LIN {X 0,Y 523.924,Z 223.222,A -85,B 0,C 180,E1 -4895.227,E2 -4895.227} C_VEL
LIN {X 0,Y 523.919,Z 223.223,A -85,B 0,C 180,E1 -4898.102,E2 -4898.102} C_VEL
LIN {X 0,Y 523.938,Z 223.222,A -85,B 0,C 180,E1 -4901.093,E2 -4901.093} C_VEL
LIN {X 0,Y 523.927,Z 223.226,A -85,B 0,C 180,E1 -4904.23,E2 -4904.23} C_VEL
LIN {X 0,Y 523.894,Z 223.223,A -85,B 0,C 180,E1 -4906.898,E2 -4906.898} C_VEL
LIN {X 0,Y 523.235,Z 223.311,A -85,B 0,C 180,E1 -4907.54,E2 -4907.54} C_VEL
LIN {X 0,Y 520.406,Z 223.66,A -85,B 0,C 180,E1 -4908.581,E2 -4908.581} C_VEL
LIN {X 0,Y 518.008,Z 223.962,A -85,B 0,C 180,E1 -4909.421,E2 -4909.421} C_VEL
LIN {X 0,Y 516.973,Z 224.088,A -85,B 0,C 180,E1 -4910.068,E2 -4910.068} C_VEL
LIN {X 0,Y 516.886,Z 224.098,A -85,B 0,C 180,E1 -4910.288,E2 -4910.288} C_VEL
LIN {X 0,Y 516.849,Z 224.105,A -85,B 0,C 180,E1 -4913.348,E2 -4913.348} C_VEL
LIN {X 0,Y 516.656,Z 224.132,A -85,B 0,C 180,E1 -4916.102,E2 -4916.102} C_VEL
LIN {X 0,Y 516.569,Z 225.057,A -85,B 0,C 180,E1 -4917.514,E2 -4917.514} C_VEL
LIN {X 0,Y 516.551,Z 227.399,A -85,B 0,C 180,E1 -4919.774,E2 -4919.774} C_VEL
LIN {X 0,Y 516.547,Z 230.185,A -85,B 0,C 180,E1 -4922.445,E2 -4922.445} C_VEL
LIN {X 0,Y 516.449,Z 232.938,A -85,B 0,C 180,E1 -4925.048,E2 -4925.048} C_VEL
LIN {X 0,Y 516.412,Z 235.802,A -85,B 0,C 180,E1 -4927.734,E2 -4927.734} C_VEL
LIN {X 0,Y 516.339,Z 239.349,A -85,B 0,C 180,E1 -4930.933,E2 -4930.933} C_VEL
LIN {X 0,Y 516.316,Z 242.204,A -85,B 0,C 180,E1 -4933.39,E2 -4933.39} C_VEL
LIN {X 0,Y 516.364,Z 245.681,A -85,B 0,C 180,E1 -4936.195,E2 -4936.195} C_VEL
LIN {X 0,Y 518.536,Z 256.766,A -85,B 0,C 180,E1 -4936.554,E2 -4936.554} C_VEL
LIN {X 0,Y 518.351,Z 269.23,A -85,B 0,C 180,E1 -4937.023,E2 -4937.023} C_VEL
LIN {X 0,Y 518.082,Z 280.828,A -85,B 0,C 180,E1 -4937.612,E2 -4937.612} C_VEL
LIN {X 0,Y 517.755,Z 292.099,A -85,B 0,C 180,E1 -4938.351,E2 -4938.351} C_VEL
LIN {X 0,Y 517.448,Z 302.758,A -85,B 0,C 180,E1 -4939.236,E2 -4939.236} C_VEL
LIN {X 0,Y 517.179,Z 312.341,A -85,B 0,C 180,E1 -4940.22,E2 -4940.22} C_VEL
LIN {X 0,Y 516.938,Z 320.187,A -85,B 0,C 180,E1 -4941.202,E2 -4941.202} C_VEL
LIN {X 0,Y 516.709,Z 327.857,A -85,B 0,C 180,E1 -4942.379,E2 -4942.379} C_VEL
LIN {X 0,Y 516.547,Z 334.883,A -85,B 0,C 180,E1 -4943.751,E2 -4943.751} C_VEL
LIN {X 0,Y 516.38,Z 339.568,A -85,B 0,C 180,E1 -4944.925,E2 -4944.925} C_VEL
LIN {X 0,Y 516.374,Z 343.149,A -85,B 0,C 180,E1 -4946.098,E2 -4946.098} C_VEL
LIN {X 0,Y 516.363,Z 345.001,A -85,B 0,C 180,E1 -4946.879,E2 -4946.879} C_VEL
LIN {X 0,Y 516.264,Z 346.404,A -85,B 0,C 180,E1 -4947.659,E2 -4947.659} C_VEL
LIN {X 0,Y 516.182,Z 348.013,A -85,B 0,C 180,E1 -4949.22,E2 -4949.22} C_VEL
LIN {X 0,Y 516.181,Z 348.249,A -85,B 0,C 180,E1 -4950,E2 -4950} C_VEL
LIN {X 0,Y 516.181,Z 348.067,A -85,B 0,C 180,E1 -4950.78,E2 -4950.78} C_VEL
LIN {X 0,Y 516.264,Z 346.529,A -85,B 0,C 180,E1 -4952.34,E2 -4952.34} C_VEL
LIN {X 0,Y 516.363,Z 345.18,A -85,B 0,C 180,E1 -4953.121,E2 -4953.121} C_VEL
LIN {X 0,Y 516.384,Z 342.34,A -85,B 0,C 180,E1 -4954.293,E2 -4954.293} C_VEL
LIN {X 0,Y 516.405,Z 338.488,A -85,B 0,C 180,E1 -4955.467,E2 -4955.467} C_VEL
LIN {X 0,Y 516.543,Z 333.377,A -85,B 0,C 180,E1 -4956.67,E2 -4956.67} C_VEL
LIN {X 0,Y 516.729,Z 327.242,A -85,B 0,C 180,E1 -4957.817,E2 -4957.817} C_VEL
LIN {X 0,Y 516.934,Z 319.392,A -85,B 0,C 180,E1 -4958.995,E2 -4958.995} C_VEL
LIN {X 0,Y 517.189,Z 311.383,A -85,B 0,C 180,E1 -4959.977,E2 -4959.977} C_VEL
LIN {X 0,Y 517.467,Z 301.605,A -85,B 0,C 180,E1 -4960.961,E2 -4960.961} C_VEL
LIN {X 0,Y 517.781,Z 291.979,A -85,B 0,C 180,E1 -4961.747,E2 -4961.747} C_VEL
LIN {X 0,Y 518.035,Z 281.52,A -85,B 0,C 180,E1 -4962.44,E2 -4962.44} C_VEL
LIN {X 0,Y 518.341,Z 269.027,A -85,B 0,C 180,E1 -4963.077,E2 -4963.077} C_VEL
LIN {X 0,Y 518.392,Z 255.726,A -85,B 0,C 180,E1 -4963.575,E2 -4963.575} C_VEL
LIN {X 0,Y 516.333,Z 245.547,A -85,B 0,C 180,E1 -4963.906,E2 -4963.906} C_VEL
LIN {X 0,Y 516.348,Z 242.346,A -85,B 0,C 180,E1 -4966.608,E2 -4966.608} C_VEL
LIN {X 0,Y 516.34,Z 239.456,A -85,B 0,C 180,E1 -4969.067,E2 -4969.067} C_VEL
LIN {X 0,Y 516.411,Z 235.882,A -85,B 0,C 180,E1 -4972.265,E2 -4972.265} C_VEL
LIN {X 0,Y 516.448,Z 232.99,A -85,B 0,C 180,E1 -4974.952,E2 -4974.952} C_VEL
LIN {X 0,Y 516.522,Z 229.994,A -85,B 0,C 180,E1 -4977.82,E2 -4977.82} C_VEL
LIN {X 0,Y 516.574,Z 226.678,A -85,B 0,C 180,E1 -4981.005,E2 -4981.005} C_VEL
LIN {X 0,Y 516.584,Z 224.643,A -85,B 0,C 180,E1 -4982.969,E2 -4982.969} C_VEL
LIN {X 0,Y 516.647,Z 224.133,A -85,B 0,C 180,E1 -4983.923,E2 -4983.923} C_VEL
LIN {X 0,Y 516.85,Z 224.105,A -85,B 0,C 180,E1 -4986.749,E2 -4986.749} C_VEL
LIN {X 0,Y 516.885,Z 224.098,A -85,B 0,C 180,E1 -4989.721,E2 -4989.721} C_VEL
LIN {X 0,Y 516.909,Z 224.096,A -85,B 0,C 180,E1 -4991.776,E2 -4991.776} C_VEL
LIN {X 0,Y 516.898,Z 224.095,A -85,B 0,C 180,E1 -4995.007,E2 -4995.007} C_VEL
LIN {X 0,Y 516.905,Z 224.096,A -85,B 0,C 180,E1 -4998.4,E2 -4998.4} C_VEL
LIN {X 0,Y 516.883,Z 224.101,A -85,B 0,C 180,E1 -5001.284,E2 -5001.284} C_VEL
LIN {X 0,Y 516.874,Z 224.104,A -85,B 0,C 180,E1 -5004.22,E2 -5004.22} C_VEL
LIN {X 0,Y 516.884,Z 224.098,A -85,B 0,C 180,E1 -5007.052,E2 -5007.052} C_VEL
LIN {X 0,Y 516.867,Z 224.102,A -85,B 0,C 180,E1 -5009.794,E2 -5009.794} C_VEL
LIN {X 0,Y 516.886,Z 224.1,A -85,B 0,C 180,E1 -5012.465,E2 -5012.465} C_VEL
LIN {X 0,Y 516.871,Z 224.101,A -85,B 0,C 180,E1 -5015.07,E2 -5015.07} C_VEL
LIN {X 0,Y 516.872,Z 224.103,A -85,B 0,C 180,E1 -5017.622,E2 -5017.622} C_VEL
LIN {X 0,Y 516.932,Z 224.093,A -85,B 0,C 180,E1 -5020.13,E2 -5020.13} C_VEL
LIN {X 0,Y 516.876,Z 224.101,A -85,B 0,C 180,E1 -5023.409,E2 -5023.409} C_VEL
LIN {X 0,Y 516.875,Z 224.099,A -85,B 0,C 180,E1 -5025.833,E2 -5025.833} C_VEL
LIN {X 0,Y 516.97,Z 224.091,A -85,B 0,C 180,E1 -5028.234,E2 -5028.234} C_VEL
LIN {X 0,Y 516.969,Z 224.092,A -85,B 0,C 180,E1 -5031.4,E2 -5031.4} C_VEL
LIN {X 0,Y 517.003,Z 224.085,A -85,B 0,C 180,E1 -5033.757,E2 -5033.757} C_VEL
LIN {X 0,Y 516.98,Z 224.09,A -85,B 0,C 180,E1 -5036.883,E2 -5036.883} C_VEL
LIN {X 0,Y 516.962,Z 224.093,A -85,B 0,C 180,E1 -5038.442,E2 -5038.442} C_VEL
LIN {X 0,Y 517.093,Z 224.073,A -85,B 0,C 180,E1 -5040.779,E2 -5040.779} C_VEL
LIN {X 0,Y 517.014,Z 224.084,A -85,B 0,C 180,E1 -5043.117,E2 -5043.117} C_VEL
LIN {X 0,Y 517.006,Z 224.084,A -85,B 0,C 180,E1 -5046.243,E2 -5046.243} C_VEL
LIN {X 0,Y 516.935,Z 224.091,A -85,B 0,C 180,E1 -5049.39,E2 -5049.39} C_VEL
LIN {X 0,Y 516.902,Z 224.097,A -85,B 0,C 180,E1 -5052.565,E2 -5052.565} C_VEL
LIN {X 0,Y 516.903,Z 224.1,A -85,B 0,C 180,E1 -5055.779,E2 -5055.779} C_VEL
LIN {X 0,Y 516.928,Z 224.093,A -85,B 0,C 180,E1 -5058.222,E2 -5058.222} C_VEL
LIN {X 0,Y 516.916,Z 224.097,A -85,B 0,C 180,E1 -5060.701,E2 -5060.701} C_VEL
LIN {X 0,Y 516.886,Z 224.103,A -85,B 0,C 180,E1 -5064.073,E2 -5064.073} C_VEL
LIN {X 0,Y 516.841,Z 224.102,A -85,B 0,C 180,E1 -5066.663,E2 -5066.663} C_VEL
LIN {X 0,Y 516.889,Z 224.101,A -85,B 0,C 180,E1 -5069.519,E2 -5069.519} C_VEL
LIN {X 0,Y 516.899,Z 224.099,A -85,B 0,C 180,E1 -5072.543,E2 -5072.543} C_VEL
LIN {X 0,Y 516.867,Z 224.101,A -85,B 0,C 180,E1 -5075.329,E2 -5075.329} C_VEL
LIN {X 0,Y 516.879,Z 224.101,A -85,B 0,C 180,E1 -5077.942,E2 -5077.942} C_VEL
LIN {X 0,Y 516.852,Z 224.102,A -85,B 0,C 180,E1 -5080.745,E2 -5080.745} C_VEL
LIN {X 0,Y 516.883,Z 224.098,A -85,B 0,C 180,E1 -5083.903,E2 -5083.903} C_VEL
LIN {X 0,Y 516.884,Z 224.103,A -85,B 0,C 180,E1 -5086.107,E2 -5086.107} C_VEL
LIN {X 0,Y 516.916,Z 224.098,A -85,B 0,C 180,E1 -5088.399,E2 -5088.399} C_VEL
LIN {X 0,Y 516.895,Z 224.105,A -85,B 0,C 180,E1 -5091.385,E2 -5091.385} C_VEL
LIN {X 0,Y 518.007,Z 230.529,A -85,B 0,C 180,E1 -5093.83,E2 -5093.83} C_VEL
LIN {X 0,Y 518.034,Z 237.244,A -85,B 0,C 180,E1 -5096.204,E2 -5096.204} C_VEL
LIN {X 0,Y 517.77,Z 245.421,A -85,B 0,C 180,E1 -5098.949,E2 -5098.949} C_VEL
LIN {X 0,Y 517.573,Z 254.625,A -85,B 0,C 180,E1 -5101.96,E2 -5101.96} C_VEL
LIN {X 0,Y 517.321,Z 262.957,A -85,B 0,C 180,E1 -5104.663,E2 -5104.663} C_VEL
LIN {X 0,Y 517.117,Z 272.225,A -85,B 0,C 180,E1 -5107.633,E2 -5107.633} C_VEL
LIN {X 0,Y 516.906,Z 281.492,A -85,B 0,C 180,E1 -5110.542,E2 -5110.542} C_VEL
LIN {X 0,Y 516.71,Z 290.759,A -85,B 0,C 180,E1 -5113.403,E2 -5113.403} C_VEL
LIN {X 0,Y 516.582,Z 299.732,A -85,B 0,C 180,E1 -5116.095,E2 -5116.095} C_VEL
LIN {X 0,Y 518.513,Z 312.183,A -85,B 0,C 180,E1 -5116.429,E2 -5116.429} C_VEL
LIN {X 0,Y 518.281,Z 324.984,A -85,B 0,C 180,E1 -5116.872,E2 -5116.872} C_VEL
LIN {X 0,Y 517.947,Z 337.175,A -85,B 0,C 180,E1 -5117.461,E2 -5117.461} C_VEL
LIN {X 0,Y 517.652,Z 347.772,A -85,B 0,C 180,E1 -5118.122,E2 -5118.122} C_VEL
LIN {X 0,Y 517.411,Z 358.262,A -85,B 0,C 180,E1 -5118.939,E2 -5118.939} C_VEL
LIN {X 0,Y 517.093,Z 367.539,A -85,B 0,C 180,E1 -5119.823,E2 -5119.823} C_VEL
LIN {X 0,Y 516.867,Z 375.991,A -85,B 0,C 180,E1 -5120.807,E2 -5120.807} C_VEL
LIN {X 0,Y 516.641,Z 384.237,A -85,B 0,C 180,E1 -5121.985,E2 -5121.985} C_VEL
LIN {X 0,Y 516.479,Z 391.077,A -85,B 0,C 180,E1 -5123.201,E2 -5123.201} C_VEL
LIN {X 0,Y 516.405,Z 396.95,A -85,B 0,C 180,E1 -5124.533,E2 -5124.533} C_VEL
LIN {X 0,Y 516.344,Z 400.895,A -85,B 0,C 180,E1 -5125.707,E2 -5125.707} C_VEL
LIN {X 0,Y 516.282,Z 403.808,A -85,B 0,C 180,E1 -5126.879,E2 -5126.879} C_VEL
LIN {X 0,Y 516.261,Z 405.197,A -85,B 0,C 180,E1 -5127.659,E2 -5127.659} C_VEL
LIN {X 0,Y 516.16,Z 406.786,A -85,B 0,C 180,E1 -5129.22,E2 -5129.22} C_VEL
LIN {X 0,Y 516.154,Z 407,A -85,B 0,C 180,E1 -5130,E2 -5130} C_VEL
LIN {X 0,Y 516.192,Z 406.185,A -85,B 0,C 180,E1 -5131.56,E2 -5131.56} C_VEL
LIN {X 0,Y 516.261,Z 405.198,A -85,B 0,C 180,E1 -5132.341,E2 -5132.341} C_VEL
LIN {X 0,Y 516.282,Z 403.81,A -85,B 0,C 180,E1 -5133.121,E2 -5133.121} C_VEL
LIN {X 0,Y 516.344,Z 400.895,A -85,B 0,C 180,E1 -5134.293,E2 -5134.293} C_VEL
LIN {X 0,Y 516.405,Z 396.948,A -85,B 0,C 180,E1 -5135.467,E2 -5135.467} C_VEL
LIN {X 0,Y 516.487,Z 391.03,A -85,B 0,C 180,E1 -5136.808,E2 -5136.808} C_VEL
LIN {X 0,Y 516.641,Z 384.236,A -85,B 0,C 180,E1 -5138.015,E2 -5138.015} C_VEL
LIN {X 0,Y 516.868,Z 375.99,A -85,B 0,C 180,E1 -5139.194,E2 -5139.194} C_VEL
LIN {X 0,Y 517.093,Z 367.537,A -85,B 0,C 180,E1 -5140.177,E2 -5140.177} C_VEL
LIN {X 0,Y 517.453,Z 357.094,A -85,B 0,C 180,E1 -5141.16,E2 -5141.16} C_VEL
LIN {X 0,Y 517.706,Z 345.73,A -85,B 0,C 180,E1 -5142.019,E2 -5142.019} C_VEL
LIN {X 0,Y 517.987,Z 335.404,A -85,B 0,C 180,E1 -5142.638,E2 -5142.638} C_VEL
LIN {X 0,Y 518.294,Z 323.758,A -85,B 0,C 180,E1 -5143.178,E2 -5143.178} C_VEL
LIN {X 0,Y 518.436,Z 310.796,A -85,B 0,C 180,E1 -5143.611,E2 -5143.611} C_VEL
LIN {X 0,Y 516.566,Z 299.529,A -85,B 0,C 180,E1 -5143.925,E2 -5143.925} C_VEL
LIN {X 0,Y 516.71,Z 290.759,A -85,B 0,C 180,E1 -5146.597,E2 -5146.597} C_VEL
LIN {X 0,Y 516.906,Z 281.491,A -85,B 0,C 180,E1 -5149.458,E2 -5149.458} C_VEL
LIN {X 0,Y 517.1,Z 271.962,A -85,B 0,C 180,E1 -5152.452,E2 -5152.452} C_VEL
LIN {X 0,Y 517.322,Z 262.957,A -85,B 0,C 180,E1 -5155.337,E2 -5155.337} C_VEL
LIN {X 0,Y 517.574,Z 254.625,A -85,B 0,C 180,E1 -5158.04,E2 -5158.04} C_VEL
LIN {X 0,Y 517.805,Z 244.879,A -85,B 0,C 180,E1 -5161.231,E2 -5161.231} C_VEL
LIN {X 0,Y 518.051,Z 236.209,A -85,B 0,C 180,E1 -5164.153,E2 -5164.153} C_VEL
LIN {X 0,Y 518.005,Z 230.494,A -85,B 0,C 180,E1 -5166.17,E2 -5166.17} C_VEL
LIN {X 0,Y 516.889,Z 224.104,A -85,B 0,C 180,E1 -5168.616,E2 -5168.616} C_VEL
LIN {X 0,Y 516.915,Z 224.101,A -85,B 0,C 180,E1 -5171.775,E2 -5171.775} C_VEL
LIN {X 0,Y 516.899,Z 224.101,A -85,B 0,C 180,E1 -5175.007,E2 -5175.007} C_VEL
LIN {X 0,Y 516.889,Z 224.098,A -85,B 0,C 180,E1 -5178.402,E2 -5178.402} C_VEL
LIN {X 0,Y 516.877,Z 224.098,A -85,B 0,C 180,E1 -5181.284,E2 -5181.284} C_VEL
LIN {X 0,Y 516.872,Z 224.104,A -85,B 0,C 180,E1 -5184.22,E2 -5184.22} C_VEL
LIN {X 0,Y 516.899,Z 224.1,A -85,B 0,C 180,E1 -5187.053,E2 -5187.053} C_VEL
LIN {X 0,Y 516.871,Z 224.1,A -85,B 0,C 180,E1 -5189.795,E2 -5189.795} C_VEL
LIN {X 0,Y 516.876,Z 224.105,A -85,B 0,C 180,E1 -5192.464,E2 -5192.464} C_VEL
LIN {X 0,Y 516.847,Z 224.102,A -85,B 0,C 180,E1 -5195.069,E2 -5195.069} C_VEL
LIN {X 0,Y 516.874,Z 224.103,A -85,B 0,C 180,E1 -5197.622,E2 -5197.622} C_VEL
LIN {X 0,Y 516.937,Z 224.092,A -85,B 0,C 180,E1 -5200.13,E2 -5200.13} C_VEL
LIN {X 0,Y 516.912,Z 224.099,A -85,B 0,C 180,E1 -5202.596,E2 -5202.596} C_VEL
LIN {X 0,Y 516.94,Z 224.092,A -85,B 0,C 180,E1 -5205.03,E2 -5205.03} C_VEL
LIN {X 0,Y 516.93,Z 224.093,A -85,B 0,C 180,E1 -5208.233,E2 -5208.233} C_VEL
LIN {X 0,Y 516.951,Z 224.095,A -85,B 0,C 180,E1 -5211.399,E2 -5211.399} C_VEL
LIN {X 0,Y 517.007,Z 224.083,A -85,B 0,C 180,E1 -5213.757,E2 -5213.757} C_VEL
LIN {X 0,Y 517.015,Z 224.084,A -85,B 0,C 180,E1 -5216.883,E2 -5216.883} C_VEL
LIN {X 0,Y 517.095,Z 224.072,A -85,B 0,C 180,E1 -5219.221,E2 -5219.221} C_VEL
LIN {X 0,Y 517.075,Z 224.073,A -85,B 0,C 180,E1 -5222.337,E2 -5222.337} C_VEL
LIN {X 0,Y 517.026,Z 224.082,A -85,B 0,C 180,E1 -5225.46,E2 -5225.46} C_VEL
LIN {X 0,Y 516.968,Z 224.089,A -85,B 0,C 180,E1 -5227.813,E2 -5227.813} C_VEL
LIN {X 0,Y 516.956,Z 224.09,A -85,B 0,C 180,E1 -5230.972,E2 -5230.972} C_VEL
LIN {X 0,Y 516.906,Z 224.1,A -85,B 0,C 180,E1 -5233.364,E2 -5233.364} C_VEL
LIN {X 0,Y 516.858,Z 224.101,A -85,B 0,C 180,E1 -5235.781,E2 -5235.781} C_VEL
LIN {X 0,Y 516.883,Z 224.098,A -85,B 0,C 180,E1 -5238.224,E2 -5238.224} C_VEL
LIN {X 0,Y 516.918,Z 224.097,A -85,B 0,C 180,E1 -5240.701,E2 -5240.701} C_VEL
LIN {X 0,Y 516.896,Z 224.101,A -85,B 0,C 180,E1 -5244.073,E2 -5244.073} C_VEL
LIN {X 0,Y 516.915,Z 224.095,A -85,B 0,C 180,E1 -5246.659,E2 -5246.659} C_VEL
LIN {X 0,Y 516.884,Z 224.098,A -85,B 0,C 180,E1 -5249.517,E2 -5249.517} C_VEL
LIN {X 0,Y 516.899,Z 224.1,A -85,B 0,C 180,E1 -5252.543,E2 -5252.543} C_VEL
LIN {X 0,Y 516.87,Z 224.101,A -85,B 0,C 180,E1 -5255.329,E2 -5255.329} C_VEL
LIN {X 0,Y 516.884,Z 224.1,A -85,B 0,C 180,E1 -5257.943,E2 -5257.943} C_VEL
LIN {X 0,Y 516.885,Z 224.103,A -85,B 0,C 180,E1 -5260.742,E2 -5260.742} C_VEL
LIN {X 0,Y 516.884,Z 224.099,A -85,B 0,C 180,E1 -5263.903,E2 -5263.903} C_VEL
LIN {X 0,Y 516.848,Z 224.101,A -85,B 0,C 180,E1 -5266.899,E2 -5266.899} C_VEL
LIN {X 0,Y 516.884,Z 224.103,A -85,B 0,C 180,E1 -5269.59,E2 -5269.59} C_VEL
LIN {X 0,Y 516.886,Z 224.098,A -85,B 0,C 180,E1 -5270.288,E2 -5270.288} C_VEL
LIN {X 0,Y 516.213,Z 224.184,A -85,B 0,C 180,E1 -5270.938,E2 -5270.938} C_VEL
LIN {X 0,Y 513.361,Z 224.539,A -85,B 0,C 180,E1 -5271.993,E2 -5271.993} C_VEL
LIN {X 0,Y 510.939,Z 224.842,A -85,B 0,C 180,E1 -5272.843,E2 -5272.843} C_VEL
LIN {X 0,Y 509.878,Z 224.972,A -85,B 0,C 180,E1 -5273.5,E2 -5273.5} C_VEL
LIN {X 0,Y 509.781,Z 224.984,A -85,B 0,C 180,E1 -5273.722,E2 -5273.722} C_VEL
LIN {X 0,Y 509.56,Z 225.014,A -85,B 0,C 180,E1 -5276.516,E2 -5276.516} C_VEL
LIN {X 0,Y 509.513,Z 227.071,A -85,B 0,C 180,E1 -5278.782,E2 -5278.782} C_VEL
LIN {X 0,Y 509.466,Z 230.42,A -85,B 0,C 180,E1 -5282.029,E2 -5282.029} C_VEL
LIN {X 0,Y 509.405,Z 233.186,A -85,B 0,C 180,E1 -5284.679,E2 -5284.679} C_VEL
LIN {X 0,Y 509.326,Z 236.28,A -85,B 0,C 180,E1 -5287.595,E2 -5287.595} C_VEL
LIN {X 0,Y 509.265,Z 239.624,A -85,B 0,C 180,E1 -5290.658,E2 -5290.658} C_VEL
LIN {X 0,Y 509.254,Z 242.514,A -85,B 0,C 180,E1 -5293.153,E2 -5293.153} C_VEL
LIN {X 0,Y 509.325,Z 246.006,A -85,B 0,C 180,E1 -5296.001,E2 -5296.001} C_VEL
LIN {X 0,Y 511.642,Z 257.212,A -85,B 0,C 180,E1 -5296.369,E2 -5296.369} C_VEL
LIN {X 0,Y 511.447,Z 269.671,A -85,B 0,C 180,E1 -5296.844,E2 -5296.844} C_VEL
LIN {X 0,Y 511.16,Z 281.811,A -85,B 0,C 180,E1 -5297.472,E2 -5297.472} C_VEL
LIN {X 0,Y 510.832,Z 292.533,A -85,B 0,C 180,E1 -5298.191,E2 -5298.191} C_VEL
LIN {X 0,Y 510.493,Z 303.191,A -85,B 0,C 180,E1 -5299.088,E2 -5299.088} C_VEL
LIN {X 0,Y 510.193,Z 312.774,A -85,B 0,C 180,E1 -5300.085,E2 -5300.085} C_VEL
LIN {X 0,Y 509.95,Z 320.618,A -85,B 0,C 180,E1 -5301.08,E2 -5301.08} C_VEL
LIN {X 0,Y 509.67,Z 328.288,A -85,B 0,C 180,E1 -5302.273,E2 -5302.273} C_VEL
LIN {X 0,Y 509.501,Z 335.312,A -85,B 0,C 180,E1 -5303.664,E2 -5303.664} C_VEL
LIN {X 0,Y 509.311,Z 339.998,A -85,B 0,C 180,E1 -5304.854,E2 -5304.854} C_VEL
LIN {X 0,Y 509.308,Z 343.578,A -85,B 0,C 180,E1 -5306.044,E2 -5306.044} C_VEL
LIN {X 0,Y 509.304,Z 345.428,A -85,B 0,C 180,E1 -5306.836,E2 -5306.836} C_VEL
LIN {X 0,Y 509.195,Z 346.831,A -85,B 0,C 180,E1 -5307.627,E2 -5307.627} C_VEL
LIN {X 0,Y 509.096,Z 348.44,A -85,B 0,C 180,E1 -5309.209,E2 -5309.209} C_VEL
LIN {X 0,Y 509.095,Z 348.676,A -85,B 0,C 180,E1 -5310,E2 -5310} C_VEL
LIN {X 0,Y 509.095,Z 348.494,A -85,B 0,C 180,E1 -5310.791,E2 -5310.791} C_VEL
LIN {X 0,Y 509.195,Z 346.954,A -85,B 0,C 180,E1 -5312.373,E2 -5312.373} C_VEL
LIN {X 0,Y 509.304,Z 345.605,A -85,B 0,C 180,E1 -5313.164,E2 -5313.164} C_VEL
LIN {X 0,Y 509.32,Z 342.765,A -85,B 0,C 180,E1 -5314.352,E2 -5314.352} C_VEL
LIN {X 0,Y 509.35,Z 338.913,A -85,B 0,C 180,E1 -5315.543,E2 -5315.543} C_VEL
LIN {X 0,Y 509.509,Z 333.083,A -85,B 0,C 180,E1 -5316.91,E2 -5316.91} C_VEL
LIN {X 0,Y 509.738,Z 326.449,A -85,B 0,C 180,E1 -5318.124,E2 -5318.124} C_VEL
LIN {X 0,Y 509.969,Z 318.344,A -85,B 0,C 180,E1 -5319.319,E2 -5319.319} C_VEL
LIN {X 0,Y 510.305,Z 310.036,A -85,B 0,C 180,E1 -5320.314,E2 -5320.314} C_VEL
LIN {X 0,Y 510.602,Z 299.779,A -85,B 0,C 180,E1 -5321.311,E2 -5321.311} C_VEL
LIN {X 0,Y 510.956,Z 288.483,A -85,B 0,C 180,E1 -5322.188,E2 -5322.188} C_VEL
LIN {X 0,Y 511.283,Z 276.667,A -85,B 0,C 180,E1 -5322.907,E2 -5322.907} C_VEL
LIN {X 0,Y 511.529,Z 264.673,A -85,B 0,C 180,E1 -5323.457,E2 -5323.457} C_VEL
LIN {X 0,Y 511.478,Z 256.521,A -85,B 0,C 180,E1 -5323.749,E2 -5323.749} C_VEL
LIN {X 0,Y 509.289,Z 245.909,A -85,B 0,C 180,E1 -5324.102,E2 -5324.102} C_VEL
LIN {X 0,Y 509.278,Z 242.62,A -85,B 0,C 180,E1 -5326.846,E2 -5326.846} C_VEL
LIN {X 0,Y 509.265,Z 239.73,A -85,B 0,C 180,E1 -5329.342,E2 -5329.342} C_VEL
LIN {X 0,Y 509.324,Z 236.364,A -85,B 0,C 180,E1 -5332.404,E2 -5332.404} C_VEL
LIN {X 0,Y 509.404,Z 233.253,A -85,B 0,C 180,E1 -5335.321,E2 -5335.321} C_VEL
LIN {X 0,Y 509.453,Z 230.472,A -85,B 0,C 180,E1 -5338.006,E2 -5338.006} C_VEL
LIN {X 0,Y 509.512,Z 227.14,A -85,B 0,C 180,E1 -5341.217,E2 -5341.217} C_VEL
LIN {X 0,Y 509.557,Z 225.015,A -85,B 0,C 180,E1 -5343.484,E2 -5343.484} C_VEL
LIN {X 0,Y 509.785,Z 224.983,A -85,B 0,C 180,E1 -5346.357,E2 -5346.357} C_VEL
LIN {X 0,Y 509.849,Z 224.977,A -85,B 0,C 180,E1 -5349.352,E2 -5349.352} C_VEL
LIN {X 0,Y 509.816,Z 224.981,A -85,B 0,C 180,E1 -5352.492,E2 -5352.492} C_VEL
LIN {X 0,Y 509.841,Z 224.976,A -85,B 0,C 180,E1 -5355.33,E2 -5355.33} C_VEL
LIN {X 0,Y 509.848,Z 224.976,A -85,B 0,C 180,E1 -5358.573,E2 -5358.573} C_VEL
LIN {X 0,Y 509.853,Z 224.975,A -85,B 0,C 180,E1 -5361.787,E2 -5361.787} C_VEL
LIN {X 0,Y 509.833,Z 224.978,A -85,B 0,C 180,E1 -5364.622,E2 -5364.622} C_VEL
LIN {X 0,Y 509.863,Z 224.976,A -85,B 0,C 180,E1 -5367.481,E2 -5367.481} C_VEL
LIN {X 0,Y 509.855,Z 224.973,A -85,B 0,C 180,E1 -5370.275,E2 -5370.275} C_VEL
LIN {X 0,Y 509.882,Z 224.971,A -85,B 0,C 180,E1 -5373.629,E2 -5373.629} C_VEL
LIN {X 0,Y 509.826,Z 224.98,A -85,B 0,C 180,E1 -5376.436,E2 -5376.436} C_VEL
LIN {X 0,Y 509.92,Z 224.968,A -85,B 0,C 180,E1 -5379.845,E2 -5379.845} C_VEL
LIN {X 0,Y 509.849,Z 224.979,A -85,B 0,C 180,E1 -5383.173,E2 -5383.173} C_VEL
LIN {X 0,Y 509.848,Z 224.974,A -85,B 0,C 180,E1 -5385.634,E2 -5385.634} C_VEL
LIN {X 0,Y 509.917,Z 224.967,A -85,B 0,C 180,E1 -5388.875,E2 -5388.875} C_VEL
LIN {X 0,Y 509.954,Z 224.963,A -85,B 0,C 180,E1 -5392.078,E2 -5392.078} C_VEL
LIN {X 0,Y 509.977,Z 224.959,A -85,B 0,C 180,E1 -5394.464,E2 -5394.464} C_VEL
LIN {X 0,Y 510.044,Z 224.948,A -85,B 0,C 180,E1 -5397.631,E2 -5397.631} C_VEL
LIN {X 0,Y 510.064,Z 224.948,A -85,B 0,C 180,E1 -5400.789,E2 -5400.789} C_VEL
LIN {X 0,Y 509.956,Z 224.964,A -85,B 0,C 180,E1 -5403.16,E2 -5403.16} C_VEL
LIN {X 0,Y 509.957,Z 224.962,A -85,B 0,C 180,E1 -5406.33,E2 -5406.33} C_VEL
LIN {X 0,Y 509.902,Z 224.972,A -85,B 0,C 180,E1 -5408.72,E2 -5408.72} C_VEL
LIN {X 0,Y 509.903,Z 224.97,A -85,B 0,C 180,E1 -5411.932,E2 -5411.932} C_VEL
LIN {X 0,Y 509.898,Z 224.97,A -85,B 0,C 180,E1 -5415.242,E2 -5415.242} C_VEL
LIN {X 0,Y 509.886,Z 224.971,A -85,B 0,C 180,E1 -5417.998,E2 -5417.998} C_VEL
LIN {X 0,Y 509.854,Z 224.977,A -85,B 0,C 180,E1 -5421.002,E2 -5421.002} C_VEL
LIN {X 0,Y 509.821,Z 224.979,A -85,B 0,C 180,E1 -5423.564,E2 -5423.564} C_VEL
LIN {X 0,Y 509.817,Z 224.978,A -85,B 0,C 180,E1 -5426.356,E2 -5426.356} C_VEL
LIN {X 0,Y 509.839,Z 224.977,A -85,B 0,C 180,E1 -5428.847,E2 -5428.847} C_VEL
LIN {X 0,Y 509.821,Z 224.979,A -85,B 0,C 180,E1 -5431.59,E2 -5431.59} C_VEL
LIN {X 0,Y 509.849,Z 224.977,A -85,B 0,C 180,E1 -5434.414,E2 -5434.414} C_VEL
LIN {X 0,Y 509.809,Z 224.981,A -85,B 0,C 180,E1 -5437.342,E2 -5437.342} C_VEL
LIN {X 0,Y 509.815,Z 224.977,A -85,B 0,C 180,E1 -5440.385,E2 -5440.385} C_VEL
LIN {X 0,Y 509.801,Z 224.985,A -85,B 0,C 180,E1 -5443.059,E2 -5443.059} C_VEL
LIN {X 0,Y 509.824,Z 224.979,A -85,B 0,C 180,E1 -5445.793,E2 -5445.793} C_VEL
LIN {X 0,Y 509.858,Z 224.977,A -85,B 0,C 180,E1 -5448.574,E2 -5448.574} C_VEL
LIN {X 0,Y 509.853,Z 225.045,A -85,B 0,C 180,E1 -5451.157,E2 -5451.157} C_VEL
LIN {X 0,Y 511.032,Z 231.69,A -85,B 0,C 180,E1 -5453.746,E2 -5453.746} C_VEL
LIN {X 0,Y 511.089,Z 237.083,A -85,B 0,C 180,E1 -5455.681,E2 -5455.681} C_VEL
LIN {X 0,Y 510.847,Z 245.392,A -85,B 0,C 180,E1 -5458.536,E2 -5458.536} C_VEL
LIN {X 0,Y 510.561,Z 255.093,A -85,B 0,C 180,E1 -5461.761,E2 -5461.761} C_VEL
LIN {X 0,Y 510.3,Z 264.281,A -85,B 0,C 180,E1 -5464.726,E2 -5464.726} C_VEL
LIN {X 0,Y 510.081,Z 273.672,A -85,B 0,C 180,E1 -5467.774,E2 -5467.774} C_VEL
LIN {X 0,Y 509.856,Z 282.816,A -85,B 0,C 180,E1 -5470.681,E2 -5470.681} C_VEL
LIN {X 0,Y 509.645,Z 293.407,A -85,B 0,C 180,E1 -5473.99,E2 -5473.99} C_VEL
LIN {X 0,Y 509.536,Z 299.731,A -85,B 0,C 180,E1 -5475.899,E2 -5475.899} C_VEL
LIN {X 0,Y 511.588,Z 312.183,A -85,B 0,C 180,E1 -5476.241,E2 -5476.241} C_VEL
LIN {X 0,Y 511.361,Z 324.984,A -85,B 0,C 180,E1 -5476.691,E2 -5476.691} C_VEL
LIN {X 0,Y 511.024,Z 337.174,A -85,B 0,C 180,E1 -5477.288,E2 -5477.288} C_VEL
LIN {X 0,Y 510.674,Z 348.197,A -85,B 0,C 180,E1 -5477.987,E2 -5477.987} C_VEL
LIN {X 0,Y 510.371,Z 359.4,A -85,B 0,C 180,E1 -5478.885,E2 -5478.885} C_VEL
LIN {X 0,Y 510.035,Z 369.335,A -85,B 0,C 180,E1 -5479.881,E2 -5479.881} C_VEL
LIN {X 0,Y 509.76,Z 378.961,A -85,B 0,C 180,E1 -5481.077,E2 -5481.077} C_VEL
LIN {X 0,Y 509.522,Z 386.622,A -85,B 0,C 180,E1 -5482.271,E2 -5482.271} C_VEL
LIN {X 0,Y 509.336,Z 393.68,A -85,B 0,C 180,E1 -5483.662,E2 -5483.662} C_VEL
LIN {X 0,Y 509.248,Z 398.373,A -85,B 0,C 180,E1 -5484.853,E2 -5484.853} C_VEL
LIN {X 0,Y 509.253,Z 401.958,A -85,B 0,C 180,E1 -5486.043,E2 -5486.043} C_VEL
LIN {X 0,Y 509.2,Z 403.808,A -85,B 0,C 180,E1 -5486.835,E2 -5486.835} C_VEL
LIN {X 0,Y 509.161,Z 405.196,A -85,B 0,C 180,E1 -5487.627,E2 -5487.627} C_VEL
LIN {X 0,Y 509.073,Z 406.786,A -85,B 0,C 180,E1 -5489.209,E2 -5489.209} C_VEL
LIN {X 0,Y 509.065,Z 407,A -85,B 0,C 180,E1 -5490,E2 -5490} C_VEL
LIN {X 0,Y 509.112,Z 406.185,A -85,B 0,C 180,E1 -5491.582,E2 -5491.582} C_VEL
LIN {X 0,Y 509.161,Z 405.198,A -85,B 0,C 180,E1 -5492.373,E2 -5492.373} C_VEL
LIN {X 0,Y 509.2,Z 403.81,A -85,B 0,C 180,E1 -5493.165,E2 -5493.165} C_VEL
LIN {X 0,Y 509.234,Z 400.895,A -85,B 0,C 180,E1 -5494.353,E2 -5494.353} C_VEL
LIN {X 0,Y 509.345,Z 396.948,A -85,B 0,C 180,E1 -5495.543,E2 -5495.543} C_VEL
LIN {X 0,Y 509.41,Z 391.281,A -85,B 0,C 180,E1 -5496.854,E2 -5496.854} C_VEL
LIN {X 0,Y 509.585,Z 384.235,A -85,B 0,C 180,E1 -5498.127,E2 -5498.127} C_VEL
LIN {X 0,Y 509.846,Z 375.99,A -85,B 0,C 180,E1 -5499.321,E2 -5499.321} C_VEL
LIN {X 0,Y 510.083,Z 367.537,A -85,B 0,C 180,E1 -5500.318,E2 -5500.318} C_VEL
LIN {X 0,Y 510.479,Z 357.093,A -85,B 0,C 180,E1 -5501.314,E2 -5501.314} C_VEL
LIN {X 0,Y 510.738,Z 346.472,A -85,B 0,C 180,E1 -5502.133,E2 -5502.133} C_VEL
LIN {X 0,Y 511.054,Z 335.404,A -85,B 0,C 180,E1 -5502.812,E2 -5502.812} C_VEL
LIN {X 0,Y 511.396,Z 323.758,A -85,B 0,C 180,E1 -5503.359,E2 -5503.359} C_VEL
LIN {X 0,Y 511.527,Z 311.71,A -85,B 0,C 180,E1 -5503.773,E2 -5503.773} C_VEL
LIN {X 0,Y 509.526,Z 299.529,A -85,B 0,C 180,E1 -5504.121,E2 -5504.121} C_VEL
LIN {X 0,Y 509.718,Z 289.435,A -85,B 0,C 180,E1 -5507.244,E2 -5507.244} C_VEL
LIN {X 0,Y 509.948,Z 279.334,A -85,B 0,C 180,E1 -5510.419,E2 -5510.419} C_VEL
LIN {X 0,Y 510.178,Z 269.576,A -85,B 0,C 180,E1 -5513.547,E2 -5513.547} C_VEL
LIN {X 0,Y 510.429,Z 260.488,A -85,B 0,C 180,E1 -5516.495,E2 -5516.495} C_VEL
LIN {X 0,Y 510.585,Z 252.003,A -85,B 0,C 180,E1 -5519.252,E2 -5519.252} C_VEL
LIN {X 0,Y 510.878,Z 243.878,A -85,B 0,C 180,E1 -5521.981,E2 -5521.981} C_VEL
LIN {X 0,Y 511.114,Z 235.729,A -85,B 0,C 180,E1 -5524.795,E2 -5524.795} C_VEL
LIN {X 0,Y 511.029,Z 231.678,A -85,B 0,C 180,E1 -5526.254,E2 -5526.254} C_VEL
LIN {X 0,Y 509.856,Z 224.979,A -85,B 0,C 180,E1 -5528.907,E2 -5528.907} C_VEL
LIN {X 0,Y 509.859,Z 224.98,A -85,B 0,C 180,E1 -5531.897,E2 -5531.897} C_VEL
LIN {X 0,Y 509.843,Z 224.978,A -85,B 0,C 180,E1 -5534.67,E2 -5534.67} C_VEL
LIN {X 0,Y 509.808,Z 224.981,A -85,B 0,C 180,E1 -5537.507,E2 -5537.507} C_VEL
LIN {X 0,Y 509.834,Z 224.981,A -85,B 0,C 180,E1 -5540.646,E2 -5540.646} C_VEL
LIN {X 0,Y 509.813,Z 224.981,A -85,B 0,C 180,E1 -5543.646,E2 -5543.646} C_VEL
LIN {X 0,Y 509.863,Z 224.973,A -85,B 0,C 180,E1 -5546.539,E2 -5546.539} C_VEL
LIN {X 0,Y 509.838,Z 224.978,A -85,B 0,C 180,E1 -5549.334,E2 -5549.334} C_VEL
LIN {X 0,Y 509.835,Z 224.977,A -85,B 0,C 180,E1 -5552.051,E2 -5552.051} C_VEL
LIN {X 0,Y 509.803,Z 224.98,A -85,B 0,C 180,E1 -5554.7,E2 -5554.7} C_VEL
LIN {X 0,Y 509.83,Z 224.979,A -85,B 0,C 180,E1 -5557.458,E2 -5557.458} C_VEL
LIN {X 0,Y 509.922,Z 224.967,A -85,B 0,C 180,E1 -5559.845,E2 -5559.845} C_VEL
LIN {X 0,Y 509.878,Z 224.973,A -85,B 0,C 180,E1 -5563.174,E2 -5563.174} C_VEL
LIN {X 0,Y 509.855,Z 224.974,A -85,B 0,C 180,E1 -5565.634,E2 -5565.634} C_VEL
LIN {X 0,Y 509.894,Z 224.971,A -85,B 0,C 180,E1 -5568.131,E2 -5568.131} C_VEL
LIN {X 0,Y 509.897,Z 224.972,A -85,B 0,C 180,E1 -5571.279,E2 -5571.279} C_VEL
LIN {X 0,Y 509.959,Z 224.962,A -85,B 0,C 180,E1 -5573.67,E2 -5573.67} C_VEL
LIN {X 0,Y 510.06,Z 224.95,A -85,B 0,C 180,E1 -5577.631,E2 -5577.631} C_VEL
LIN {X 0,Y 510.038,Z 224.954,A -85,B 0,C 180,E1 -5580,E2 -5580} C_VEL
LIN {X 0,Y 510.046,Z 224.948,A -85,B 0,C 180,E1 -5582.369,E2 -5582.369} C_VEL
LIN {X 0,Y 509.956,Z 224.963,A -85,B 0,C 180,E1 -5586.33,E2 -5586.33} C_VEL
LIN {X 0,Y 509.909,Z 224.971,A -85,B 0,C 180,E1 -5588.72,E2 -5588.72} C_VEL
LIN {X 0,Y 509.91,Z 224.97,A -85,B 0,C 180,E1 -5591.932,E2 -5591.932} C_VEL
LIN {X 0,Y 509.9,Z 224.973,A -85,B 0,C 180,E1 -5595.242,E2 -5595.242} C_VEL
LIN {X 0,Y 509.843,Z 224.977,A -85,B 0,C 180,E1 -5598.485,E2 -5598.485} C_VEL
LIN {X 0,Y 509.856,Z 224.975,A -85,B 0,C 180,E1 -5601.002,E2 -5601.002} C_VEL
LIN {X 0,Y 509.828,Z 224.98,A -85,B 0,C 180,E1 -5603.564,E2 -5603.564} C_VEL
LIN {X 0,Y 509.911,Z 224.967,A -85,B 0,C 180,E1 -5606.377,E2 -5606.377} C_VEL
LIN {X 0,Y 509.83,Z 224.976,A -85,B 0,C 180,E1 -5609.753,E2 -5609.753} C_VEL
LIN {X 0,Y 509.871,Z 224.973,A -85,B 0,C 180,E1 -5612.773,E2 -5612.773} C_VEL
LIN {X 0,Y 509.83,Z 224.979,A -85,B 0,C 180,E1 -5615.578,E2 -5615.578} C_VEL
LIN {X 0,Y 509.854,Z 224.975,A -85,B 0,C 180,E1 -5618.338,E2 -5618.338} C_VEL
LIN {X 0,Y 509.855,Z 224.975,A -85,B 0,C 180,E1 -5621.426,E2 -5621.426} C_VEL
LIN {X 0,Y 509.843,Z 224.976,A -85,B 0,C 180,E1 -5624.67,E2 -5624.67} C_VEL
LIN {X 0,Y 509.848,Z 224.977,A -85,B 0,C 180,E1 -5628.105,E2 -5628.105} C_VEL
LIN {X 0,Y 509.85,Z 224.976,A -85,B 0,C 180,E1 -5630.647,E2 -5630.647} C_VEL
LIN {X 0,Y 509.788,Z 224.983,A -85,B 0,C 180,E1 -5633.643,E2 -5633.643} C_VEL
LIN {X 0,Y 509.781,Z 224.984,A -85,B 0,C 180,E1 -5633.722,E2 -5633.722} C_VEL
LIN {X 0,Y 509.064,Z 225.096,A -85,B 0,C 180,E1 -5634.382,E2 -5634.382} C_VEL
LIN {X 0,Y 506.114,Z 225.445,A -85,B 0,C 180,E1 -5635.452,E2 -5635.452} C_VEL
LIN {X 0,Y 503.631,Z 225.753,A -85,B 0,C 180,E1 -5636.313,E2 -5636.313} C_VEL
LIN {X 0,Y 502.551,Z 225.984,A -85,B 0,C 180,E1 -5636.977,E2 -5636.977} C_VEL
LIN {X 0,Y 502.455,Z 226.166,A -85,B 0,C 180,E1 -5637.201,E2 -5637.201} C_VEL
LIN {X 0,Y 502.428,Z 229.16,A -85,B 0,C 180,E1 -5640.142,E2 -5640.142} C_VEL
LIN {X 0,Y 502.363,Z 231.604,A -85,B 0,C 180,E1 -5642.505,E2 -5642.505} C_VEL
LIN {X 0,Y 502.292,Z 234.649,A -85,B 0,C 180,E1 -5645.433,E2 -5645.433} C_VEL
LIN {X 0,Y 502.253,Z 237.144,A -85,B 0,C 180,E1 -5647.802,E2 -5647.802} C_VEL
LIN {X 0,Y 502.212,Z 239.931,A -85,B 0,C 180,E1 -5650.375,E2 -5650.375} C_VEL
LIN {X 0,Y 502.214,Z 242.826,A -85,B 0,C 180,E1 -5652.91,E2 -5652.91} C_VEL
LIN {X 0,Y 502.227,Z 246.326,A -85,B 0,C 180,E1 -5655.799,E2 -5655.799} C_VEL
LIN {X 0,Y 504.767,Z 258.416,A -85,B 0,C 180,E1 -5656.206,E2 -5656.206} C_VEL
LIN {X 0,Y 504.558,Z 271.235,A -85,B 0,C 180,E1 -5656.713,E2 -5656.713} C_VEL
LIN {X 0,Y 504.254,Z 282.668,A -85,B 0,C 180,E1 -5657.323,E2 -5657.323} C_VEL
LIN {X 0,Y 503.86,Z 294.25,A -85,B 0,C 180,E1 -5658.127,E2 -5658.127} C_VEL
LIN {X 0,Y 503.519,Z 304.685,A -85,B 0,C 180,E1 -5659.037,E2 -5659.037} C_VEL
LIN {X 0,Y 503.222,Z 313.206,A -85,B 0,C 180,E1 -5659.946,E2 -5659.946} C_VEL
LIN {X 0,Y 502.949,Z 321.049,A -85,B 0,C 180,E1 -5660.955,E2 -5660.955} C_VEL
LIN {X 0,Y 502.642,Z 328.719,A -85,B 0,C 180,E1 -5662.165,E2 -5662.165} C_VEL
LIN {X 0,Y 502.455,Z 335.742,A -85,B 0,C 180,E1 -5663.575,E2 -5663.575} C_VEL
LIN {X 0,Y 502.244,Z 340.428,A -85,B 0,C 180,E1 -5664.781,E2 -5664.781} C_VEL
LIN {X 0,Y 502.245,Z 344.006,A -85,B 0,C 180,E1 -5665.988,E2 -5665.988} C_VEL
LIN {X 0,Y 502.246,Z 345.855,A -85,B 0,C 180,E1 -5666.791,E2 -5666.791} C_VEL
LIN {X 0,Y 502.13,Z 347.258,A -85,B 0,C 180,E1 -5667.593,E2 -5667.593} C_VEL
LIN {X 0,Y 502.011,Z 348.867,A -85,B 0,C 180,E1 -5669.198,E2 -5669.198} C_VEL
LIN {X 0,Y 502.008,Z 349.103,A -85,B 0,C 180,E1 -5670,E2 -5670} C_VEL
LIN {X 0,Y 502.011,Z 348.92,A -85,B 0,C 180,E1 -5670.802,E2 -5670.802} C_VEL
LIN {X 0,Y 502.13,Z 347.379,A -85,B 0,C 180,E1 -5672.406,E2 -5672.406} C_VEL
LIN {X 0,Y 502.247,Z 346.03,A -85,B 0,C 180,E1 -5673.209,E2 -5673.209} C_VEL
LIN {X 0,Y 502.259,Z 343.19,A -85,B 0,C 180,E1 -5674.414,E2 -5674.414} C_VEL
LIN {X 0,Y 502.297,Z 339.337,A -85,B 0,C 180,E1 -5675.621,E2 -5675.621} C_VEL
LIN {X 0,Y 502.478,Z 333.7,A -85,B 0,C 180,E1 -5676.968,E2 -5676.968} C_VEL
LIN {X 0,Y 502.707,Z 326.873,A -85,B 0,C 180,E1 -5678.239,E2 -5678.239} C_VEL
LIN {X 0,Y 502.968,Z 318.766,A -85,B 0,C 180,E1 -5679.45,E2 -5679.45} C_VEL
LIN {X 0,Y 503.347,Z 310.457,A -85,B 0,C 180,E1 -5680.458,E2 -5680.458} C_VEL
LIN {X 0,Y 503.668,Z 300.198,A -85,B 0,C 180,E1 -5681.469,E2 -5681.469} C_VEL
LIN {X 0,Y 504.02,Z 289.386,A -85,B 0,C 180,E1 -5682.324,E2 -5682.324} C_VEL
LIN {X 0,Y 504.36,Z 278.892,A -85,B 0,C 180,E1 -5682.985,E2 -5682.985} C_VEL
LIN {X 0,Y 504.638,Z 266.377,A -85,B 0,C 180,E1 -5683.592,E2 -5683.592} C_VEL
LIN {X 0,Y 504.558,Z 257.311,A -85,B 0,C 180,E1 -5683.928,E2 -5683.928} C_VEL
LIN {X 0,Y 502.223,Z 246.264,A -85,B 0,C 180,E1 -5684.305,E2 -5684.305} C_VEL
LIN {X 0,Y 502.231,Z 242.933,A -85,B 0,C 180,E1 -5687.089,E2 -5687.089} C_VEL
LIN {X 0,Y 502.243,Z 239.212,A -85,B 0,C 180,E1 -5690.356,E2 -5690.356} C_VEL
LIN {X 0,Y 502.25,Z 236.302,A -85,B 0,C 180,E1 -5693.067,E2 -5693.067} C_VEL
LIN {X 0,Y 502.325,Z 233.517,A -85,B 0,C 180,E1 -5695.704,E2 -5695.704} C_VEL
LIN {X 0,Y 502.401,Z 230.746,A -85,B 0,C 180,E1 -5698.4,E2 -5698.4} C_VEL
LIN {X 0,Y 502.466,Z 227.641,A -85,B 0,C 180,E1 -5701.437,E2 -5701.437} C_VEL
LIN {X 0,Y 502.464,Z 225.998,A -85,B 0,C 180,E1 -5703.059,E2 -5703.059} C_VEL
LIN {X 0,Y 502.739,Z 225.863,A -85,B 0,C 180,E1 -5705.954,E2 -5705.954} C_VEL
LIN {X 0,Y 502.804,Z 225.855,A -85,B 0,C 180,E1 -5708.976,E2 -5708.976} C_VEL
LIN {X 0,Y 502.806,Z 225.857,A -85,B 0,C 180,E1 -5712.199,E2 -5712.199} C_VEL
LIN {X 0,Y 502.788,Z 225.855,A -85,B 0,C 180,E1 -5715.47,E2 -5715.47} C_VEL
LIN {X 0,Y 502.797,Z 225.855,A -85,B 0,C 180,E1 -5717.861,E2 -5717.861} C_VEL
LIN {X 0,Y 502.802,Z 225.855,A -85,B 0,C 180,E1 -5721.024,E2 -5721.024} C_VEL
LIN {X 0,Y 502.778,Z 225.86,A -85,B 0,C 180,E1 -5724.169,E2 -5724.169} C_VEL
LIN {X 0,Y 502.833,Z 225.848,A -85,B 0,C 180,E1 -5726.994,E2 -5726.994} C_VEL
LIN {X 0,Y 502.812,Z 225.851,A -85,B 0,C 180,E1 -5730.066,E2 -5730.066} C_VEL
LIN {X 0,Y 502.847,Z 225.848,A -85,B 0,C 180,E1 -5733.444,E2 -5733.444} C_VEL
LIN {X 0,Y 502.779,Z 225.858,A -85,B 0,C 180,E1 -5736.085,E2 -5736.085} C_VEL
LIN {X 0,Y 502.787,Z 225.855,A -85,B 0,C 180,E1 -5738.689,E2 -5738.689} C_VEL
LIN {X 0,Y 502.815,Z 225.855,A -85,B 0,C 180,E1 -5741.248,E2 -5741.248} C_VEL
LIN {X 0,Y 502.838,Z 225.851,A -85,B 0,C 180,E1 -5744.665,E2 -5744.665} C_VEL
LIN {X 0,Y 502.88,Z 225.845,A -85,B 0,C 180,E1 -5748.039,E2 -5748.039} C_VEL
LIN {X 0,Y 502.875,Z 225.846,A -85,B 0,C 180,E1 -5751.157,E2 -5751.157} C_VEL
LIN {X 0,Y 502.908,Z 225.841,A -85,B 0,C 180,E1 -5753.581,E2 -5753.581} C_VEL
LIN {X 0,Y 502.868,Z 225.849,A -85,B 0,C 180,E1 -5756.795,E2 -5756.795} C_VEL
LIN {X 0,Y 502.9,Z 225.844,A -85,B 0,C 180,E1 -5758.398,E2 -5758.398} C_VEL
LIN {X 0,Y 503.014,Z 225.827,A -85,B 0,C 180,E1 -5760.801,E2 -5760.801} C_VEL
LIN {X 0,Y 502.899,Z 225.843,A -85,B 0,C 180,E1 -5763.204,E2 -5763.204} C_VEL
LIN {X 0,Y 502.91,Z 225.84,A -85,B 0,C 180,E1 -5766.419,E2 -5766.419} C_VEL
LIN {X 0,Y 502.861,Z 225.847,A -85,B 0,C 180,E1 -5768.844,E2 -5768.844} C_VEL
LIN {X 0,Y 502.845,Z 225.852,A -85,B 0,C 180,E1 -5772.102,E2 -5772.102} C_VEL
LIN {X 0,Y 502.852,Z 225.848,A -85,B 0,C 180,E1 -5775.4,E2 -5775.4} C_VEL
LIN {X 0,Y 502.844,Z 225.848,A -85,B 0,C 180,E1 -5778.12,E2 -5778.12} C_VEL
LIN {X 0,Y 502.832,Z 225.852,A -85,B 0,C 180,E1 -5780.536,E2 -5780.536} C_VEL
LIN {X 0,Y 502.789,Z 225.854,A -85,B 0,C 180,E1 -5783.041,E2 -5783.041} C_VEL
LIN {X 0,Y 502.778,Z 225.859,A -85,B 0,C 180,E1 -5785.679,E2 -5785.679} C_VEL
LIN {X 0,Y 502.775,Z 225.855,A -85,B 0,C 180,E1 -5788.377,E2 -5788.377} C_VEL
LIN {X 0,Y 502.795,Z 225.858,A -85,B 0,C 180,E1 -5791.143,E2 -5791.143} C_VEL
LIN {X 0,Y 502.806,Z 225.855,A -85,B 0,C 180,E1 -5793.994,E2 -5793.994} C_VEL
LIN {X 0,Y 502.766,Z 225.858,A -85,B 0,C 180,E1 -5797.176,E2 -5797.176} C_VEL
LIN {X 0,Y 502.772,Z 225.855,A -85,B 0,C 180,E1 -5800.017,E2 -5800.017} C_VEL
LIN {X 0,Y 502.773,Z 225.855,A -85,B 0,C 180,E1 -5802.195,E2 -5802.195} C_VEL
LIN {X 0,Y 502.788,Z 225.855,A -85,B 0,C 180,E1 -5805.47,E2 -5805.47} C_VEL
LIN {X 0,Y 502.822,Z 225.852,A -85,B 0,C 180,E1 -5808.934,E2 -5808.934} C_VEL
LIN {X 0,Y 502.818,Z 225.93,A -85,B 0,C 180,E1 -5810.896,E2 -5810.896} C_VEL
LIN {X 0,Y 504.008,Z 232.701,A -85,B 0,C 180,E1 -5813.601,E2 -5813.601} C_VEL
LIN {X 0,Y 504.111,Z 238.544,A -85,B 0,C 180,E1 -5815.724,E2 -5815.724} C_VEL
LIN {X 0,Y 503.774,Z 247.738,A -85,B 0,C 180,E1 -5818.924,E2 -5818.924} C_VEL
LIN {X 0,Y 503.508,Z 257.283,A -85,B 0,C 180,E1 -5822.122,E2 -5822.122} C_VEL
LIN {X 0,Y 503.276,Z 265.479,A -85,B 0,C 180,E1 -5824.792,E2 -5824.792} C_VEL
LIN {X 0,Y 503.026,Z 274.872,A -85,B 0,C 180,E1 -5827.838,E2 -5827.838} C_VEL
LIN {X 0,Y 502.8,Z 284.14,A -85,B 0,C 180,E1 -5830.824,E2 -5830.824} C_VEL
LIN {X 0,Y 502.561,Z 294.731,A -85,B 0,C 180,E1 -5834.175,E2 -5834.175} C_VEL
LIN {X 0,Y 502.482,Z 299.582,A -85,B 0,C 180,E1 -5835.693,E2 -5835.693} C_VEL
LIN {X 0,Y 504.688,Z 313.096,A -85,B 0,C 180,E1 -5836.075,E2 -5836.075} C_VEL
LIN {X 0,Y 504.424,Z 326.112,A -85,B 0,C 180,E1 -5836.556,E2 -5836.556} C_VEL
LIN {X 0,Y 504.036,Z 338.643,A -85,B 0,C 180,E1 -5837.194,E2 -5837.194} C_VEL
LIN {X 0,Y 503.694,Z 349.589,A -85,B 0,C 180,E1 -5837.919,E2 -5837.919} C_VEL
LIN {X 0,Y 503.359,Z 360.47,A -85,B 0,C 180,E1 -5838.83,E2 -5838.83} C_VEL
LIN {X 0,Y 503.032,Z 369.334,A -85,B 0,C 180,E1 -5839.739,E2 -5839.739} C_VEL
LIN {X 0,Y 502.704,Z 378.961,A -85,B 0,C 180,E1 -5840.951,E2 -5840.951} C_VEL
LIN {X 0,Y 502.47,Z 386.622,A -85,B 0,C 180,E1 -5842.162,E2 -5842.162} C_VEL
LIN {X 0,Y 502.275,Z 393.68,A -85,B 0,C 180,E1 -5843.573,E2 -5843.573} C_VEL
LIN {X 0,Y 502.185,Z 398.373,A -85,B 0,C 180,E1 -5844.781,E2 -5844.781} C_VEL
LIN {X 0,Y 502.151,Z 401.958,A -85,B 0,C 180,E1 -5845.987,E2 -5845.987} C_VEL
LIN {X 0,Y 502.121,Z 403.808,A -85,B 0,C 180,E1 -5846.791,E2 -5846.791} C_VEL
LIN {X 0,Y 502.066,Z 405.195,A -85,B 0,C 180,E1 -5847.593,E2 -5847.593} C_VEL
LIN {X 0,Y 501.99,Z 406.786,A -85,B 0,C 180,E1 -5849.198,E2 -5849.198} C_VEL
LIN {X 0,Y 501.98,Z 407,A -85,B 0,C 180,E1 -5850,E2 -5850} C_VEL
LIN {X 0,Y 502.036,Z 406.185,A -85,B 0,C 180,E1 -5851.605,E2 -5851.605} C_VEL
LIN {X 0,Y 502.066,Z 405.197,A -85,B 0,C 180,E1 -5852.407,E2 -5852.407} C_VEL
LIN {X 0,Y 502.121,Z 403.81,A -85,B 0,C 180,E1 -5853.21,E2 -5853.21} C_VEL
LIN {X 0,Y 502.128,Z 400.895,A -85,B 0,C 180,E1 -5854.415,E2 -5854.415} C_VEL
LIN {X 0,Y 502.26,Z 396.948,A -85,B 0,C 180,E1 -5855.621,E2 -5855.621} C_VEL
LIN {X 0,Y 502.336,Z 390.976,A -85,B 0,C 180,E1 -5857.012,E2 -5857.012} C_VEL
LIN {X 0,Y 502.542,Z 384.235,A -85,B 0,C 180,E1 -5858.242,E2 -5858.242} C_VEL
LIN {X 0,Y 502.811,Z 375.99,A -85,B 0,C 180,E1 -5859.453,E2 -5859.453} C_VEL
LIN {X 0,Y 503.077,Z 367.537,A -85,B 0,C 180,E1 -5860.464,E2 -5860.464} C_VEL
LIN {X 0,Y 503.505,Z 357.092,A -85,B 0,C 180,E1 -5861.473,E2 -5861.473} C_VEL
LIN {X 0,Y 503.799,Z 345.382,A -85,B 0,C 180,E1 -5862.381,E2 -5862.381} C_VEL
LIN {X 0,Y 504.172,Z 333.485,A -85,B 0,C 180,E1 -5863.092,E2 -5863.092} C_VEL
LIN {X 0,Y 504.541,Z 321.161,A -85,B 0,C 180,E1 -5863.647,E2 -5863.647} C_VEL
LIN {X 0,Y 504.546,Z 312.167,A -85,B 0,C 180,E1 -5863.955,E2 -5863.955} C_VEL
LIN {X 0,Y 502.465,Z 299.529,A -85,B 0,C 180,E1 -5864.324,E2 -5864.324} C_VEL
LIN {X 0,Y 502.663,Z 289.435,A -85,B 0,C 180,E1 -5867.494,E2 -5867.494} C_VEL
LIN {X 0,Y 502.905,Z 279.828,A -85,B 0,C 180,E1 -5870.558,E2 -5870.558} C_VEL
LIN {X 0,Y 503.188,Z 269.576,A -85,B 0,C 180,E1 -5873.894,E2 -5873.894} C_VEL
LIN {X 0,Y 503.454,Z 259.907,A -85,B 0,C 180,E1 -5877.012,E2 -5877.012} C_VEL
LIN {X 0,Y 503.724,Z 250.436,A -85,B 0,C 180,E1 -5880.151,E2 -5880.151} C_VEL
LIN {X 0,Y 504.012,Z 241.57,A -85,B 0,C 180,E1 -5883.212,E2 -5883.212} C_VEL
LIN {X 0,Y 504.168,Z 234.188,A -85,B 0,C 180,E1 -5885.837,E2 -5885.837} C_VEL
LIN {X 0,Y 503.335,Z 228.864,A -85,B 0,C 180,E1 -5887.906,E2 -5887.906} C_VEL
LIN {X 0,Y 502.802,Z 225.857,A -85,B 0,C 180,E1 -5889.17,E2 -5889.17} C_VEL
LIN {X 0,Y 502.807,Z 225.858,A -85,B 0,C 180,E1 -5892.199,E2 -5892.199} C_VEL
LIN {X 0,Y 502.789,Z 225.859,A -85,B 0,C 180,E1 -5895.47,E2 -5895.47} C_VEL
LIN {X 0,Y 502.798,Z 225.852,A -85,B 0,C 180,E1 -5897.861,E2 -5897.861} C_VEL
LIN {X 0,Y 502.795,Z 225.854,A -85,B 0,C 180,E1 -5901.023,E2 -5901.023} C_VEL
LIN {X 0,Y 502.775,Z 225.86,A -85,B 0,C 180,E1 -5904.17,E2 -5904.17} C_VEL
LIN {X 0,Y 502.837,Z 225.851,A -85,B 0,C 180,E1 -5906.994,E2 -5906.994} C_VEL
LIN {X 0,Y 502.814,Z 225.851,A -85,B 0,C 180,E1 -5910.066,E2 -5910.066} C_VEL
LIN {X 0,Y 502.777,Z 225.854,A -85,B 0,C 180,E1 -5913.46,E2 -5913.46} C_VEL
LIN {X 0,Y 502.771,Z 225.861,A -85,B 0,C 180,E1 -5916.085,E2 -5916.085} C_VEL
LIN {X 0,Y 502.788,Z 225.855,A -85,B 0,C 180,E1 -5918.689,E2 -5918.689} C_VEL
LIN {X 0,Y 502.832,Z 225.852,A -85,B 0,C 180,E1 -5921.248,E2 -5921.248} C_VEL
LIN {X 0,Y 502.854,Z 225.848,A -85,B 0,C 180,E1 -5924.6,E2 -5924.6} C_VEL
LIN {X 0,Y 502.874,Z 225.847,A -85,B 0,C 180,E1 -5928.043,E2 -5928.043} C_VEL
LIN {X 0,Y 502.856,Z 225.848,A -85,B 0,C 180,E1 -5931.156,E2 -5931.156} C_VEL
LIN {X 0,Y 502.911,Z 225.84,A -85,B 0,C 180,E1 -5933.581,E2 -5933.581} C_VEL
LIN {X 0,Y 502.9,Z 225.843,A -85,B 0,C 180,E1 -5936.796,E2 -5936.796} C_VEL
LIN {X 0,Y 503.015,Z 225.826,A -85,B 0,C 180,E1 -5939.199,E2 -5939.199} C_VEL
LIN {X 0,Y 503.015,Z 225.824,A -85,B 0,C 180,E1 -5942.402,E2 -5942.402} C_VEL
LIN {X 0,Y 502.933,Z 225.837,A -85,B 0,C 180,E1 -5945.614,E2 -5945.614} C_VEL
LIN {X 0,Y 502.886,Z 225.845,A -85,B 0,C 180,E1 -5948.034,E2 -5948.034} C_VEL
LIN {X 0,Y 502.882,Z 225.844,A -85,B 0,C 180,E1 -5951.283,E2 -5951.283} C_VEL
LIN {X 0,Y 502.83,Z 225.849,A -85,B 0,C 180,E1 -5954.571,E2 -5954.571} C_VEL
LIN {X 0,Y 502.806,Z 225.85,A -85,B 0,C 180,E1 -5957.909,E2 -5957.909} C_VEL
LIN {X 0,Y 502.834,Z 225.853,A -85,B 0,C 180,E1 -5960.536,E2 -5960.536} C_VEL
LIN {X 0,Y 502.793,Z 225.854,A -85,B 0,C 180,E1 -5963.041,E2 -5963.041} C_VEL
LIN {X 0,Y 502.824,Z 225.852,A -85,B 0,C 180,E1 -5965.677,E2 -5965.677} C_VEL
LIN {X 0,Y 502.777,Z 225.856,A -85,B 0,C 180,E1 -5968.377,E2 -5968.377} C_VEL
LIN {X 0,Y 502.795,Z 225.851,A -85,B 0,C 180,E1 -5971.498,E2 -5971.498} C_VEL
LIN {X 0,Y 502.794,Z 225.856,A -85,B 0,C 180,E1 -5973.995,E2 -5973.995} C_VEL
LIN {X 0,Y 502.782,Z 225.857,A -85,B 0,C 180,E1 -5977.178,E2 -5977.178} C_VEL
LIN {X 0,Y 502.791,Z 225.854,A -85,B 0,C 180,E1 -5980.015,E2 -5980.015} C_VEL
LIN {X 0,Y 502.807,Z 225.854,A -85,B 0,C 180,E1 -5982.199,E2 -5982.199} C_VEL
LIN {X 0,Y 502.789,Z 225.853,A -85,B 0,C 180,E1 -5985.47,E2 -5985.47} C_VEL
LIN {X 0,Y 502.798,Z 225.858,A -85,B 0,C 180,E1 -5987.86,E2 -5987.86} C_VEL
LIN {X 0,Y 502.805,Z 225.854,A -85,B 0,C 180,E1 -5991.024,E2 -5991.024} C_VEL
LIN {X 0,Y 502.74,Z 225.863,A -85,B 0,C 180,E1 -5994.175,E2 -5994.175} C_VEL
LIN {X 0,Y 502.465,Z 226.02,A -85,B 0,C 180,E1 -5997.059,E2 -5997.059} C_VEL
LIN {X 0,Y 502.455,Z 226.166,A -85,B 0,C 180,E1 -5997.201,E2 -5997.201} C_VEL
LIN {X 0,Y 501.764,Z 226.917,A -85,B 0,C 180,E1 -5997.865,E2 -5997.865} C_VEL
LIN {X 0,Y 498.887,Z 228.292,A -85,B 0,C 180,E1 -5998.939,E2 -5998.939} C_VEL
LIN {X 0,Y 496.461,Z 229.412,A -85,B 0,C 180,E1 -5999.805,E2 -5999.805} C_VEL
LIN {X 0,Y 495.414,Z 230.199,A -85,B 0,C 180,E1 -6000.475,E2 -6000.475} C_VEL
LIN {X 0,Y 495.324,Z 230.441,A -85,B 0,C 180,E1 -6000.702,E2 -6000.702} C_VEL
LIN {X 0,Y 495.279,Z 233.179,A -85,B 0,C 180,E1 -6003.377,E2 -6003.377} C_VEL
LIN {X 0,Y 495.218,Z 235.59,A -85,B 0,C 180,E1 -6005.697,E2 -6005.697} C_VEL
LIN {X 0,Y 495.161,Z 238.367,A -85,B 0,C 180,E1 -6008.344,E2 -6008.344} C_VEL
LIN {X 0,Y 495.145,Z 241.209,A -85,B 0,C 180,E1 -6010.946,E2 -6010.946} C_VEL
LIN {X 0,Y 495.106,Z 244.155,A -85,B 0,C 180,E1 -6013.507,E2 -6013.507} C_VEL
LIN {X 0,Y 495.167,Z 246.705,A -85,B 0,C 180,E1 -6015.592,E2 -6015.592} C_VEL
LIN {X 0,Y 497.799,Z 258.867,A -85,B 0,C 180,E1 -6016.009,E2 -6016.009} C_VEL
LIN {X 0,Y 497.682,Z 271.674,A -85,B 0,C 180,E1 -6016.526,E2 -6016.526} C_VEL
LIN {X 0,Y 497.352,Z 283.497,A -85,B 0,C 180,E1 -6017.17,E2 -6017.17} C_VEL
LIN {X 0,Y 496.943,Z 294.684,A -85,B 0,C 180,E1 -6017.959,E2 -6017.959} C_VEL
LIN {X 0,Y 496.561,Z 305.118,A -85,B 0,C 180,E1 -6018.881,E2 -6018.881} C_VEL
LIN {X 0,Y 496.236,Z 313.639,A -85,B 0,C 180,E1 -6019.803,E2 -6019.803} C_VEL
LIN {X 0,Y 495.945,Z 321.481,A -85,B 0,C 180,E1 -6020.826,E2 -6020.826} C_VEL
LIN {X 0,Y 495.629,Z 329.149,A -85,B 0,C 180,E1 -6022.053,E2 -6022.053} C_VEL
LIN {X 0,Y 495.42,Z 336.171,A -85,B 0,C 180,E1 -6023.483,E2 -6023.483} C_VEL
LIN {X 0,Y 495.179,Z 340.857,A -85,B 0,C 180,E1 -6024.707,E2 -6024.707} C_VEL
LIN {X 0,Y 495.185,Z 344.434,A -85,B 0,C 180,E1 -6025.931,E2 -6025.931} C_VEL
LIN {X 0,Y 495.191,Z 346.282,A -85,B 0,C 180,E1 -6026.745,E2 -6026.745} C_VEL
LIN {X 0,Y 495.067,Z 347.684,A -85,B 0,C 180,E1 -6027.559,E2 -6027.559} C_VEL
LIN {X 0,Y 494.93,Z 349.294,A -85,B 0,C 180,E1 -6029.186,E2 -6029.186} C_VEL
LIN {X 0,Y 494.925,Z 349.529,A -85,B 0,C 180,E1 -6030,E2 -6030} C_VEL
LIN {X 0,Y 494.929,Z 349.346,A -85,B 0,C 180,E1 -6030.814,E2 -6030.814} C_VEL
LIN {X 0,Y 495.067,Z 347.804,A -85,B 0,C 180,E1 -6032.441,E2 -6032.441} C_VEL
LIN {X 0,Y 495.191,Z 346.454,A -85,B 0,C 180,E1 -6033.254,E2 -6033.254} C_VEL
LIN {X 0,Y 495.2,Z 343.615,A -85,B 0,C 180,E1 -6034.477,E2 -6034.477} C_VEL
LIN {X 0,Y 495.248,Z 339.762,A -85,B 0,C 180,E1 -6035.701,E2 -6035.701} C_VEL
LIN {X 0,Y 495.413,Z 334.784,A -85,B 0,C 180,E1 -6036.925,E2 -6036.925} C_VEL
LIN {X 0,Y 495.651,Z 328.513,A -85,B 0,C 180,E1 -6038.152,E2 -6038.152} C_VEL
LIN {X 0,Y 495.959,Z 320.657,A -85,B 0,C 180,E1 -6039.379,E2 -6039.379} C_VEL
LIN {X 0,Y 496.299,Z 312.645,A -85,B 0,C 180,E1 -6040.402,E2 -6040.402} C_VEL
LIN {X 0,Y 496.634,Z 302.864,A -85,B 0,C 180,E1 -6041.427,E2 -6041.427} C_VEL
LIN {X 0,Y 497.012,Z 292.246,A -85,B 0,C 180,E1 -6042.321,E2 -6042.321} C_VEL
LIN {X 0,Y 497.403,Z 281.064,A -85,B 0,C 180,E1 -6043.066,E2 -6043.066} C_VEL
LIN {X 0,Y 497.724,Z 269.138,A -85,B 0,C 180,E1 -6043.681,E2 -6043.681} C_VEL
LIN {X 0,Y 497.726,Z 258.476,A -85,B 0,C 180,E1 -6044.098,E2 -6044.098} C_VEL
LIN {X 0,Y 495.149,Z 246.639,A -85,B 0,C 180,E1 -6044.513,E2 -6044.513} C_VEL
LIN {X 0,Y 495.155,Z 243.274,A -85,B 0,C 180,E1 -6047.341,E2 -6047.341} C_VEL
LIN {X 0,Y 495.169,Z 239.718,A -85,B 0,C 180,E1 -6050.487,E2 -6050.487} C_VEL
LIN {X 0,Y 495.19,Z 236.595,A -85,B 0,C 180,E1 -6053.415,E2 -6053.415} C_VEL
LIN {X 0,Y 495.267,Z 233.788,A -85,B 0,C 180,E1 -6056.098,E2 -6056.098} C_VEL
LIN {X 0,Y 495.319,Z 230.987,A -85,B 0,C 180,E1 -6058.844,E2 -6058.844} C_VEL
LIN {X 0,Y 495.414,Z 228.118,A -85,B 0,C 180,E1 -6061.661,E2 -6061.661} C_VEL
LIN {X 0,Y 495.428,Z 226.776,A -85,B 0,C 180,E1 -6063.179,E2 -6063.179} C_VEL
LIN {X 0,Y 495.688,Z 226.74,A -85,B 0,C 180,E1 -6066.083,E2 -6066.083} C_VEL
LIN {X 0,Y 495.766,Z 226.732,A -85,B 0,C 180,E1 -6068.768,E2 -6068.768} C_VEL
LIN {X 0,Y 495.753,Z 226.731,A -85,B 0,C 180,E1 -6071.782,E2 -6071.782} C_VEL
LIN {X 0,Y 495.739,Z 226.731,A -85,B 0,C 180,E1 -6075.141,E2 -6075.141} C_VEL
LIN {X 0,Y 495.752,Z 226.731,A -85,B 0,C 180,E1 -6078.218,E2 -6078.218} C_VEL
LIN {X 0,Y 495.752,Z 226.733,A -85,B 0,C 180,E1 -6081.408,E2 -6081.408} C_VEL
LIN {X 0,Y 495.75,Z 226.733,A -85,B 0,C 180,E1 -6084.462,E2 -6084.462} C_VEL
LIN {X 0,Y 495.769,Z 226.731,A -85,B 0,C 180,E1 -6087.406,E2 -6087.406} C_VEL
LIN {X 0,Y 495.759,Z 226.729,A -85,B 0,C 180,E1 -6090.253,E2 -6090.253} C_VEL
LIN {X 0,Y 495.776,Z 226.73,A -85,B 0,C 180,E1 -6093.262,E2 -6093.262} C_VEL
LIN {X 0,Y 495.727,Z 226.736,A -85,B 0,C 180,E1 -6095.724,E2 -6095.724} C_VEL
LIN {X 0,Y 495.746,Z 226.733,A -85,B 0,C 180,E1 -6098.371,E2 -6098.371} C_VEL
LIN {X 0,Y 495.775,Z 226.729,A -85,B 0,C 180,E1 -6100.971,E2 -6100.971} C_VEL
LIN {X 0,Y 495.825,Z 226.723,A -85,B 0,C 180,E1 -6104.55,E2 -6104.55} C_VEL
LIN {X 0,Y 495.832,Z 226.723,A -85,B 0,C 180,E1 -6107.965,E2 -6107.965} C_VEL
LIN {X 0,Y 495.844,Z 226.721,A -85,B 0,C 180,E1 -6111.03,E2 -6111.03} C_VEL
LIN {X 0,Y 495.862,Z 226.719,A -85,B 0,C 180,E1 -6113.489,E2 -6113.489} C_VEL
LIN {X 0,Y 495.814,Z 226.728,A -85,B 0,C 180,E1 -6116.75,E2 -6116.75} C_VEL
LIN {X 0,Y 495.87,Z 226.719,A -85,B 0,C 180,E1 -6118.376,E2 -6118.376} C_VEL
LIN {X 0,Y 495.965,Z 226.705,A -85,B 0,C 180,E1 -6120.812,E2 -6120.812} C_VEL
LIN {X 0,Y 495.997,Z 226.702,A -85,B 0,C 180,E1 -6122.436,E2 -6122.436} C_VEL
LIN {X 0,Y 495.893,Z 226.716,A -85,B 0,C 180,E1 -6125.693,E2 -6125.693} C_VEL
LIN {X 0,Y 495.838,Z 226.721,A -85,B 0,C 180,E1 -6128.149,E2 -6128.149} C_VEL
LIN {X 0,Y 495.824,Z 226.72,A -85,B 0,C 180,E1 -6131.446,E2 -6131.446} C_VEL
LIN {X 0,Y 495.783,Z 226.727,A -85,B 0,C 180,E1 -6134.783,E2 -6134.783} C_VEL
LIN {X 0,Y 495.784,Z 226.729,A -85,B 0,C 180,E1 -6137.319,E2 -6137.319} C_VEL
LIN {X 0,Y 495.774,Z 226.729,A -85,B 0,C 180,E1 -6139.89,E2 -6139.89} C_VEL
LIN {X 0,Y 495.761,Z 226.73,A -85,B 0,C 180,E1 -6142.86,E2 -6142.86} C_VEL
LIN {X 0,Y 495.718,Z 226.736,A -85,B 0,C 180,E1 -6146.072,E2 -6146.072} C_VEL
LIN {X 0,Y 495.73,Z 226.734,A -85,B 0,C 180,E1 -6148.818,E2 -6148.818} C_VEL
LIN {X 0,Y 495.757,Z 226.731,A -85,B 0,C 180,E1 -6151.725,E2 -6151.725} C_VEL
LIN {X 0,Y 495.771,Z 226.731,A -85,B 0,C 180,E1 -6154.694,E2 -6154.694} C_VEL
LIN {X 0,Y 495.723,Z 226.739,A -85,B 0,C 180,E1 -6157.562,E2 -6157.562} C_VEL
LIN {X 0,Y 495.744,Z 226.731,A -85,B 0,C 180,E1 -6160.045,E2 -6160.045} C_VEL
LIN {X 0,Y 495.707,Z 226.741,A -85,B 0,C 180,E1 -6162.885,E2 -6162.885} C_VEL
LIN {X 0,Y 495.73,Z 226.737,A -85,B 0,C 180,E1 -6165.998,E2 -6165.998} C_VEL
LIN {X 0,Y 495.768,Z 226.731,A -85,B 0,C 180,E1 -6169.3,E2 -6169.3} C_VEL
LIN {X 0,Y 495.777,Z 226.853,A -85,B 0,C 180,E1 -6170.646,E2 -6170.646} C_VEL
LIN {X 0,Y 497.039,Z 234.019,A -85,B 0,C 180,E1 -6173.568,E2 -6173.568} C_VEL
LIN {X 0,Y 497.123,Z 239.42,A -85,B 0,C 180,E1 -6175.563,E2 -6175.563} C_VEL
LIN {X 0,Y 496.832,Z 247.546,A -85,B 0,C 180,E1 -6178.44,E2 -6178.44} C_VEL
LIN {X 0,Y 496.558,Z 256.029,A -85,B 0,C 180,E1 -6181.344,E2 -6181.344} C_VEL
LIN {X 0,Y 496.308,Z 263.875,A -85,B 0,C 180,E1 -6183.961,E2 -6183.961} C_VEL
LIN {X 0,Y 496.094,Z 272.077,A -85,B 0,C 180,E1 -6186.63,E2 -6186.63} C_VEL
LIN {X 0,Y 495.841,Z 281.554,A -85,B 0,C 180,E1 -6189.701,E2 -6189.701} C_VEL
LIN {X 0,Y 495.592,Z 290.759,A -85,B 0,C 180,E1 -6192.674,E2 -6192.674} C_VEL
LIN {X 0,Y 495.412,Z 299.582,A -85,B 0,C 180,E1 -6195.485,E2 -6195.485} C_VEL
LIN {X 0,Y 497.671,Z 313.096,A -85,B 0,C 180,E1 -6195.875,E2 -6195.875} C_VEL
LIN {X 0,Y 497.506,Z 326.112,A -85,B 0,C 180,E1 -6196.365,E2 -6196.365} C_VEL
LIN {X 0,Y 497.107,Z 338.778,A -85,B 0,C 180,E1 -6197.021,E2 -6197.021} C_VEL
LIN {X 0,Y 496.718,Z 349.589,A -85,B 0,C 180,E1 -6197.747,E2 -6197.747} C_VEL
LIN {X 0,Y 496.383,Z 360.469,A -85,B 0,C 180,E1 -6198.671,E2 -6198.671} C_VEL
LIN {X 0,Y 496.006,Z 369.334,A -85,B 0,C 180,E1 -6199.592,E2 -6199.592} C_VEL
LIN {X 0,Y 495.673,Z 378.961,A -85,B 0,C 180,E1 -6200.822,E2 -6200.822} C_VEL
LIN {X 0,Y 495.403,Z 386.622,A -85,B 0,C 180,E1 -6202.05,E2 -6202.05} C_VEL
LIN {X 0,Y 495.204,Z 393.68,A -85,B 0,C 180,E1 -6203.481,E2 -6203.481} C_VEL
LIN {X 0,Y 495.123,Z 398.373,A -85,B 0,C 180,E1 -6204.706,E2 -6204.706} C_VEL
LIN {X 0,Y 495.049,Z 401.959,A -85,B 0,C 180,E1 -6205.93,E2 -6205.93} C_VEL
LIN {X 0,Y 495.043,Z 403.807,A -85,B 0,C 180,E1 -6206.745,E2 -6206.745} C_VEL
LIN {X 0,Y 494.961,Z 406.183,A -85,B 0,C 180,E1 -6208.373,E2 -6208.373} C_VEL
LIN {X 0,Y 494.898,Z 407,A -85,B 0,C 180,E1 -6210,E2 -6210} C_VEL
LIN {X 0,Y 494.961,Z 406.184,A -85,B 0,C 180,E1 -6211.627,E2 -6211.627} C_VEL
LIN {X 0,Y 495.043,Z 403.81,A -85,B 0,C 180,E1 -6213.256,E2 -6213.256} C_VEL
LIN {X 0,Y 495.029,Z 400.895,A -85,B 0,C 180,E1 -6214.479,E2 -6214.479} C_VEL
LIN {X 0,Y 495.211,Z 395.802,A -85,B 0,C 180,E1 -6215.999,E2 -6215.999} C_VEL
LIN {X 0,Y 495.278,Z 389.868,A -85,B 0,C 180,E1 -6217.337,E2 -6217.337} C_VEL
LIN {X 0,Y 495.557,Z 383.002,A -85,B 0,C 180,E1 -6218.564,E2 -6218.564} C_VEL
LIN {X 0,Y 495.856,Z 374.411,A -85,B 0,C 180,E1 -6219.793,E2 -6219.793} C_VEL
LIN {X 0,Y 496.198,Z 365.597,A -85,B 0,C 180,E1 -6220.817,E2 -6220.817} C_VEL
LIN {X 0,Y 496.581,Z 354.742,A -85,B 0,C 180,E1 -6221.842,E2 -6221.842} C_VEL
LIN {X 0,Y 496.898,Z 344.175,A -85,B 0,C 180,E1 -6222.638,E2 -6222.638} C_VEL
LIN {X 0,Y 497.246,Z 333.484,A -85,B 0,C 180,E1 -6223.278,E2 -6223.278} C_VEL
LIN {X 0,Y 497.637,Z 321.16,A -85,B 0,C 180,E1 -6223.84,E2 -6223.84} C_VEL
LIN {X 0,Y 497.587,Z 312.623,A -85,B 0,C 180,E1 -6224.141,E2 -6224.141} C_VEL
LIN {X 0,Y 495.424,Z 299.529,A -85,B 0,C 180,E1 -6224.532,E2 -6224.532} C_VEL
LIN {X 0,Y 495.638,Z 289.435,A -85,B 0,C 180,E1 -6227.75,E2 -6227.75} C_VEL
LIN {X 0,Y 495.886,Z 280.167,A -85,B 0,C 180,E1 -6230.752,E2 -6230.752} C_VEL
LIN {X 0,Y 496.121,Z 270.701,A -85,B 0,C 180,E1 -6233.812,E2 -6233.812} C_VEL
LIN {X 0,Y 496.419,Z 261.133,A -85,B 0,C 180,E1 -6236.939,E2 -6236.939} C_VEL
LIN {X 0,Y 496.735,Z 251.053,A -85,B 0,C 180,E1 -6240.339,E2 -6240.339} C_VEL
LIN {X 0,Y 497.057,Z 242.134,A -85,B 0,C 180,E1 -6243.466,E2 -6243.466} C_VEL
LIN {X 0,Y 497.197,Z 235.531,A -85,B 0,C 180,E1 -6245.855,E2 -6245.855} C_VEL
LIN {X 0,Y 496.344,Z 230.06,A -85,B 0,C 180,E1 -6248.02,E2 -6248.02} C_VEL
LIN {X 0,Y 495.746,Z 226.736,A -85,B 0,C 180,E1 -6249.413,E2 -6249.413} C_VEL
LIN {X 0,Y 495.76,Z 226.736,A -85,B 0,C 180,E1 -6251.781,E2 -6251.781} C_VEL
LIN {X 0,Y 495.741,Z 226.738,A -85,B 0,C 180,E1 -6255.141,E2 -6255.141} C_VEL
LIN {X 0,Y 495.746,Z 226.731,A -85,B 0,C 180,E1 -6258.218,E2 -6258.218} C_VEL
LIN {X 0,Y 495.747,Z 226.73,A -85,B 0,C 180,E1 -6261.408,E2 -6261.408} C_VEL
LIN {X 0,Y 495.749,Z 226.733,A -85,B 0,C 180,E1 -6264.462,E2 -6264.462} C_VEL
LIN {X 0,Y 495.772,Z 226.73,A -85,B 0,C 180,E1 -6267.406,E2 -6267.406} C_VEL
LIN {X 0,Y 495.761,Z 226.731,A -85,B 0,C 180,E1 -6270.253,E2 -6270.253} C_VEL
LIN {X 0,Y 495.742,Z 226.73,A -85,B 0,C 180,E1 -6273.271,E2 -6273.271} C_VEL
LIN {X 0,Y 495.743,Z 226.732,A -85,B 0,C 180,E1 -6276.612,E2 -6276.612} C_VEL
LIN {X 0,Y 495.784,Z 226.729,A -85,B 0,C 180,E1 -6279.324,E2 -6279.324} C_VEL
LIN {X 0,Y 495.786,Z 226.727,A -85,B 0,C 180,E1 -6281.829,E2 -6281.829} C_VEL
LIN {X 0,Y 495.829,Z 226.724,A -85,B 0,C 180,E1 -6284.549,E2 -6284.549} C_VEL
LIN {X 0,Y 495.826,Z 226.725,A -85,B 0,C 180,E1 -6287.969,E2 -6287.969} C_VEL
LIN {X 0,Y 495.81,Z 226.725,A -85,B 0,C 180,E1 -6291.03,E2 -6291.03} C_VEL
LIN {X 0,Y 495.866,Z 226.719,A -85,B 0,C 180,E1 -6293.49,E2 -6293.49} C_VEL
LIN {X 0,Y 495.844,Z 226.722,A -85,B 0,C 180,E1 -6296.75,E2 -6296.75} C_VEL
LIN {X 0,Y 495.871,Z 226.718,A -85,B 0,C 180,E1 -6298.376,E2 -6298.376} C_VEL
LIN {X 0,Y 495.976,Z 226.705,A -85,B 0,C 180,E1 -6300,E2 -6300} C_VEL
LIN {X 0,Y 495.984,Z 226.7,A -85,B 0,C 180,E1 -6302.436,E2 -6302.436} C_VEL
LIN {X 0,Y 495.889,Z 226.714,A -85,B 0,C 180,E1 -6305.694,E2 -6305.694} C_VEL
LIN {X 0,Y 495.842,Z 226.722,A -85,B 0,C 180,E1 -6308.149,E2 -6308.149} C_VEL
LIN {X 0,Y 495.857,Z 226.72,A -85,B 0,C 180,E1 -6311.445,E2 -6311.445} C_VEL
LIN {X 0,Y 495.781,Z 226.728,A -85,B 0,C 180,E1 -6314.783,E2 -6314.783} C_VEL
LIN {X 0,Y 495.776,Z 226.727,A -85,B 0,C 180,E1 -6318.235,E2 -6318.235} C_VEL
LIN {X 0,Y 495.78,Z 226.73,A -85,B 0,C 180,E1 -6320.756,E2 -6320.756} C_VEL
LIN {X 0,Y 495.748,Z 226.734,A -85,B 0,C 180,E1 -6323.387,E2 -6323.387} C_VEL
LIN {X 0,Y 495.777,Z 226.729,A -85,B 0,C 180,E1 -6326.069,E2 -6326.069} C_VEL
LIN {X 0,Y 495.726,Z 226.739,A -85,B 0,C 180,E1 -6328.818,E2 -6328.818} C_VEL
LIN {X 0,Y 495.757,Z 226.728,A -85,B 0,C 180,E1 -6331.725,E2 -6331.725} C_VEL
LIN {X 0,Y 495.767,Z 226.729,A -85,B 0,C 180,E1 -6334.693,E2 -6334.693} C_VEL
LIN {X 0,Y 495.733,Z 226.736,A -85,B 0,C 180,E1 -6337.562,E2 -6337.562} C_VEL
LIN {X 0,Y 495.762,Z 226.73,A -85,B 0,C 180,E1 -6340.047,E2 -6340.047} C_VEL
LIN {X 0,Y 495.719,Z 226.736,A -85,B 0,C 180,E1 -6342.884,E2 -6342.884} C_VEL
LIN {X 0,Y 495.727,Z 226.738,A -85,B 0,C 180,E1 -6345.998,E2 -6345.998} C_VEL
LIN {X 0,Y 495.74,Z 226.732,A -85,B 0,C 180,E1 -6348.709,E2 -6348.709} C_VEL
LIN {X 0,Y 495.754,Z 226.735,A -85,B 0,C 180,E1 -6351.408,E2 -6351.408} C_VEL
LIN {X 0,Y 495.664,Z 226.745,A -85,B 0,C 180,E1 -6354.455,E2 -6354.455} C_VEL
LIN {X 0,Y 495.403,Z 226.963,A -85,B 0,C 180,E1 -6357.185,E2 -6357.185} C_VEL
LIN {X 0,Y 495.36,Z 229.949,A -85,B 0,C 180,E1 -6360.226,E2 -6360.226} C_VEL
LIN {X 0,Y 495.324,Z 230.441,A -85,B 0,C 180,E1 -6360.702,E2 -6360.702} C_VEL
LIN {X 0,Y 494.637,Z 231.202,A -85,B 0,C 180,E1 -6361.375,E2 -6361.375} C_VEL
LIN {X 0,Y 491.741,Z 232.597,A -85,B 0,C 180,E1 -6362.465,E2 -6362.465} C_VEL
LIN {X 0,Y 489.305,Z 233.732,A -85,B 0,C 180,E1 -6363.343,E2 -6363.343} C_VEL
LIN {X 0,Y 488.267,Z 234.535,A -85,B 0,C 180,E1 -6364.023,E2 -6364.023} C_VEL
LIN {X 0,Y 488.187,Z 234.785,A -85,B 0,C 180,E1 -6364.253,E2 -6364.253} C_VEL
LIN {X 0,Y 488.15,Z 237.758,A -85,B 0,C 180,E1 -6367.135,E2 -6367.135} C_VEL
LIN {X 0,Y 488.096,Z 240.579,A -85,B 0,C 180,E1 -6369.783,E2 -6369.783} C_VEL
LIN {X 0,Y 488.104,Z 243.518,A -85,B 0,C 180,E1 -6372.4,E2 -6372.4} C_VEL
LIN {X 0,Y 488.114,Z 247.141,A -85,B 0,C 180,E1 -6375.379,E2 -6375.379} C_VEL
LIN {X 0,Y 490.968,Z 260.064,A -85,B 0,C 180,E1 -6375.836,E2 -6375.836} C_VEL
LIN {X 0,Y 490.792,Z 272.113,A -85,B 0,C 180,E1 -6376.333,E2 -6376.333} C_VEL
LIN {X 0,Y 490.474,Z 283.455,A -85,B 0,C 180,E1 -6376.956,E2 -6376.956} C_VEL
LIN {X 0,Y 490.026,Z 295.116,A -85,B 0,C 180,E1 -6377.787,E2 -6377.787} C_VEL
LIN {X 0,Y 489.619,Z 305.55,A -85,B 0,C 180,E1 -6378.722,E2 -6378.722} C_VEL
LIN {X 0,Y 489.271,Z 314.07,A -85,B 0,C 180,E1 -6379.656,E2 -6379.656} C_VEL
LIN {X 0,Y 488.955,Z 321.912,A -85,B 0,C 180,E1 -6380.694,E2 -6380.694} C_VEL
LIN {X 0,Y 488.608,Z 329.579,A -85,B 0,C 180,E1 -6381.938,E2 -6381.938} C_VEL
LIN {X 0,Y 488.359,Z 336.602,A -85,B 0,C 180,E1 -6383.389,E2 -6383.389} C_VEL
LIN {X 0,Y 488.117,Z 341.287,A -85,B 0,C 180,E1 -6384.63,E2 -6384.63} C_VEL
LIN {X 0,Y 488.128,Z 344.861,A -85,B 0,C 180,E1 -6385.872,E2 -6385.872} C_VEL
LIN {X 0,Y 488.12,Z 346.71,A -85,B 0,C 180,E1 -6386.698,E2 -6386.698} C_VEL
LIN {X 0,Y 488.007,Z 348.111,A -85,B 0,C 180,E1 -6387.524,E2 -6387.524} C_VEL
LIN {X 0,Y 487.852,Z 349.721,A -85,B 0,C 180,E1 -6389.174,E2 -6389.174} C_VEL
LIN {X 0,Y 487.844,Z 349.956,A -85,B 0,C 180,E1 -6390,E2 -6390} C_VEL
LIN {X 0,Y 487.851,Z 349.772,A -85,B 0,C 180,E1 -6390.825,E2 -6390.825} C_VEL
LIN {X 0,Y 488.006,Z 348.229,A -85,B 0,C 180,E1 -6392.476,E2 -6392.476} C_VEL
LIN {X 0,Y 488.121,Z 346.879,A -85,B 0,C 180,E1 -6393.302,E2 -6393.302} C_VEL
LIN {X 0,Y 488.141,Z 344.04,A -85,B 0,C 180,E1 -6394.542,E2 -6394.542} C_VEL
LIN {X 0,Y 488.202,Z 340.186,A -85,B 0,C 180,E1 -6395.783,E2 -6395.783} C_VEL
LIN {X 0,Y 488.383,Z 335.208,A -85,B 0,C 180,E1 -6397.025,E2 -6397.025} C_VEL
LIN {X 0,Y 488.645,Z 328.935,A -85,B 0,C 180,E1 -6398.269,E2 -6398.269} C_VEL
LIN {X 0,Y 488.952,Z 321.081,A -85,B 0,C 180,E1 -6399.514,E2 -6399.514} C_VEL
LIN {X 0,Y 489.417,Z 311.299,A -85,B 0,C 180,E1 -6400.759,E2 -6400.759} C_VEL
LIN {X 0,Y 489.801,Z 301.037,A -85,B 0,C 180,E1 -6401.798,E2 -6401.798} C_VEL
LIN {X 0,Y 490.211,Z 290.101,A -85,B 0,C 180,E1 -6402.685,E2 -6402.685} C_VEL
LIN {X 0,Y 490.56,Z 279.726,A -85,B 0,C 180,E1 -6403.357,E2 -6403.357} C_VEL
LIN {X 0,Y 490.887,Z 267.201,A -85,B 0,C 180,E1 -6403.981,E2 -6403.981} C_VEL
LIN {X 0,Y 490.81,Z 259.269,A -85,B 0,C 180,E1 -6404.287,E2 -6404.287} C_VEL
LIN {X 0,Y 488.097,Z 247.028,A -85,B 0,C 180,E1 -6404.728,E2 -6404.728} C_VEL
LIN {X 0,Y 488.096,Z 243.013,A -85,B 0,C 180,E1 -6408.135,E2 -6408.135} C_VEL
LIN {X 0,Y 488.095,Z 239.713,A -85,B 0,C 180,E1 -6411.098,E2 -6411.098} C_VEL
LIN {X 0,Y 488.117,Z 236.888,A -85,B 0,C 180,E1 -6413.775,E2 -6413.775} C_VEL
LIN {X 0,Y 488.222,Z 234.061,A -85,B 0,C 180,E1 -6416.503,E2 -6416.503} C_VEL
LIN {X 0,Y 488.268,Z 231.236,A -85,B 0,C 180,E1 -6419.3,E2 -6419.3} C_VEL
LIN {X 0,Y 488.317,Z 228.347,A -85,B 0,C 180,E1 -6422.176,E2 -6422.176} C_VEL
LIN {X 0,Y 488.424,Z 227.647,A -85,B 0,C 180,E1 -6423.428,E2 -6423.428} C_VEL
LIN {X 0,Y 488.657,Z 227.616,A -85,B 0,C 180,E1 -6426.35,E2 -6426.35} C_VEL
LIN {X 0,Y 488.704,Z 227.61,A -85,B 0,C 180,E1 -6429.254,E2 -6429.254} C_VEL
LIN {X 0,Y 488.69,Z 227.612,A -85,B 0,C 180,E1 -6432.526,E2 -6432.526} C_VEL
LIN {X 0,Y 488.703,Z 227.608,A -85,B 0,C 180,E1 -6435.197,E2 -6435.197} C_VEL
LIN {X 0,Y 488.694,Z 227.611,A -85,B 0,C 180,E1 -6438.583,E2 -6438.583} C_VEL
LIN {X 0,Y 488.705,Z 227.611,A -85,B 0,C 180,E1 -6440.948,E2 -6440.948} C_VEL
LIN {X 0,Y 488.68,Z 227.614,A -85,B 0,C 180,E1 -6443.868,E2 -6443.868} C_VEL
LIN {X 0,Y 488.738,Z 227.604,A -85,B 0,C 180,E1 -6446.877,E2 -6446.877} C_VEL
LIN {X 0,Y 488.72,Z 227.608,A -85,B 0,C 180,E1 -6449.78,E2 -6449.78} C_VEL
LIN {X 0,Y 488.726,Z 227.61,A -85,B 0,C 180,E1 -6453.072,E2 -6453.072} C_VEL
LIN {X 0,Y 488.714,Z 227.608,A -85,B 0,C 180,E1 -6455.352,E2 -6455.352} C_VEL
LIN {X 0,Y 488.702,Z 227.611,A -85,B 0,C 180,E1 -6458.043,E2 -6458.043} C_VEL
LIN {X 0,Y 488.739,Z 227.604,A -85,B 0,C 180,E1 -6460.686,E2 -6460.686} C_VEL
LIN {X 0,Y 488.756,Z 227.601,A -85,B 0,C 180,E1 -6464.145,E2 -6464.145} C_VEL
LIN {X 0,Y 488.741,Z 227.605,A -85,B 0,C 180,E1 -6467.543,E2 -6467.543} C_VEL
LIN {X 0,Y 488.768,Z 227.603,A -85,B 0,C 180,E1 -6470.064,E2 -6470.064} C_VEL
LIN {X 0,Y 488.871,Z 227.589,A -85,B 0,C 180,E1 -6472.723,E2 -6472.723} C_VEL
LIN {X 0,Y 488.802,Z 227.6,A -85,B 0,C 180,E1 -6475.051,E2 -6475.051} C_VEL
LIN {X 0,Y 488.95,Z 227.576,A -85,B 0,C 180,E1 -6477.529,E2 -6477.529} C_VEL
LIN {X 0,Y 488.916,Z 227.583,A -85,B 0,C 180,E1 -6480.824,E2 -6480.824} C_VEL
LIN {X 0,Y 488.964,Z 227.578,A -85,B 0,C 180,E1 -6482.471,E2 -6482.471} C_VEL
LIN {X 0,Y 488.851,Z 227.593,A -85,B 0,C 180,E1 -6485.776,E2 -6485.776} C_VEL
LIN {X 0,Y 488.786,Z 227.6,A -85,B 0,C 180,E1 -6488.267,E2 -6488.267} C_VEL
LIN {X 0,Y 488.786,Z 227.598,A -85,B 0,C 180,E1 -6491.613,E2 -6491.613} C_VEL
LIN {X 0,Y 488.759,Z 227.603,A -85,B 0,C 180,E1 -6495,E2 -6495} C_VEL
LIN {X 0,Y 488.758,Z 227.604,A -85,B 0,C 180,E1 -6498.442,E2 -6498.442} C_VEL
LIN {X 0,Y 488.71,Z 227.61,A -85,B 0,C 180,E1 -6501.071,E2 -6501.071} C_VEL
LIN {X 0,Y 488.672,Z 227.615,A -85,B 0,C 180,E1 -6503.747,E2 -6503.747} C_VEL
LIN {X 0,Y 488.699,Z 227.608,A -85,B 0,C 180,E1 -6506.922,E2 -6506.922} C_VEL
LIN {X 0,Y 488.721,Z 227.607,A -85,B 0,C 180,E1 -6510.22,E2 -6510.22} C_VEL
LIN {X 0,Y 488.737,Z 227.606,A -85,B 0,C 180,E1 -6513.484,E2 -6513.484} C_VEL
LIN {X 0,Y 488.675,Z 227.613,A -85,B 0,C 180,E1 -6516.353,E2 -6516.353} C_VEL
LIN {X 0,Y 488.694,Z 227.613,A -85,B 0,C 180,E1 -6519.255,E2 -6519.255} C_VEL
LIN {X 0,Y 488.669,Z 227.615,A -85,B 0,C 180,E1 -6522.528,E2 -6522.528} C_VEL
LIN {X 0,Y 488.703,Z 227.61,A -85,B 0,C 180,E1 -6525.197,E2 -6525.197} C_VEL
LIN {X 0,Y 488.709,Z 227.613,A -85,B 0,C 180,E1 -6528.4,E2 -6528.4} C_VEL
LIN {X 0,Y 488.741,Z 227.681,A -85,B 0,C 180,E1 -6530.349,E2 -6530.349} C_VEL
LIN {X 0,Y 490.041,Z 235.093,A -85,B 0,C 180,E1 -6533.431,E2 -6533.431} C_VEL
LIN {X 0,Y 490.176,Z 239.236,A -85,B 0,C 180,E1 -6535.005,E2 -6535.005} C_VEL
LIN {X 0,Y 489.894,Z 247.353,A -85,B 0,C 180,E1 -6537.94,E2 -6537.94} C_VEL
LIN {X 0,Y 489.562,Z 256.501,A -85,B 0,C 180,E1 -6541.128,E2 -6541.128} C_VEL
LIN {X 0,Y 489.26,Z 265.017,A -85,B 0,C 180,E1 -6544.016,E2 -6544.016} C_VEL
LIN {X 0,Y 488.992,Z 273.745,A -85,B 0,C 180,E1 -6546.903,E2 -6546.903} C_VEL
LIN {X 0,Y 488.786,Z 282.785,A -85,B 0,C 180,E1 -6549.813,E2 -6549.813} C_VEL
LIN {X 0,Y 488.508,Z 292.083,A -85,B 0,C 180,E1 -6552.847,E2 -6552.847} C_VEL
LIN {X 0,Y 488.372,Z 299.582,A -85,B 0,C 180,E1 -6555.271,E2 -6555.271} C_VEL
LIN {X 0,Y 490.651,Z 313.096,A -85,B 0,C 180,E1 -6555.668,E2 -6555.668} C_VEL
LIN {X 0,Y 490.836,Z 317.742,A -85,B 0,C 180,E1 -6555.833,E2 -6555.833} C_VEL
LIN {X 0,Y 490.452,Z 330.511,A -85,B 0,C 180,E1 -6556.376,E2 -6556.376} C_VEL
LIN {X 0,Y 490.04,Z 342.136,A -85,B 0,C 180,E1 -6557.046,E2 -6557.046} C_VEL
LIN {X 0,Y 489.698,Z 352.195,A -85,B 0,C 180,E1 -6557.779,E2 -6557.779} C_VEL
LIN {X 0,Y 489.322,Z 362.606,A -85,B 0,C 180,E1 -6558.715,E2 -6558.715} C_VEL
LIN {X 0,Y 488.954,Z 371.114,A -85,B 0,C 180,E1 -6559.65,E2 -6559.65} C_VEL
LIN {X 0,Y 488.657,Z 378.961,A -85,B 0,C 180,E1 -6560.689,E2 -6560.689} C_VEL
LIN {X 0,Y 488.361,Z 386.622,A -85,B 0,C 180,E1 -6561.934,E2 -6561.934} C_VEL
LIN {X 0,Y 488.141,Z 393.68,A -85,B 0,C 180,E1 -6563.386,E2 -6563.386} C_VEL
LIN {X 0,Y 488.06,Z 398.373,A -85,B 0,C 180,E1 -6564.629,E2 -6564.629} C_VEL
LIN {X 0,Y 487.947,Z 401.958,A -85,B 0,C 180,E1 -6565.87,E2 -6565.87} C_VEL
LIN {X 0,Y 487.966,Z 403.807,A -85,B 0,C 180,E1 -6566.697,E2 -6566.697} C_VEL
LIN {X 0,Y 487.889,Z 406.183,A -85,B 0,C 180,E1 -6568.349,E2 -6568.349} C_VEL
LIN {X 0,Y 487.819,Z 407,A -85,B 0,C 180,E1 -6570,E2 -6570} C_VEL
LIN {X 0,Y 487.889,Z 406.184,A -85,B 0,C 180,E1 -6571.651,E2 -6571.651} C_VEL
LIN {X 0,Y 487.967,Z 403.81,A -85,B 0,C 180,E1 -6573.303,E2 -6573.303} C_VEL
LIN {X 0,Y 487.938,Z 400.895,A -85,B 0,C 180,E1 -6574.544,E2 -6574.544} C_VEL
LIN {X 0,Y 488.105,Z 396.948,A -85,B 0,C 180,E1 -6575.785,E2 -6575.785} C_VEL
LIN {X 0,Y 488.191,Z 390.875,A -85,B 0,C 180,E1 -6577.237,E2 -6577.237} C_VEL
LIN {X 0,Y 488.454,Z 384.235,A -85,B 0,C 180,E1 -6578.481,E2 -6578.481} C_VEL
LIN {X 0,Y 488.762,Z 375.99,A -85,B 0,C 180,E1 -6579.727,E2 -6579.727} C_VEL
LIN {X 0,Y 489.09,Z 367.538,A -85,B 0,C 180,E1 -6580.767,E2 -6580.767} C_VEL
LIN {X 0,Y 489.538,Z 357.09,A -85,B 0,C 180,E1 -6581.805,E2 -6581.805} C_VEL
LIN {X 0,Y 489.898,Z 345.847,A -85,B 0,C 180,E1 -6582.704,E2 -6582.704} C_VEL
LIN {X 0,Y 490.262,Z 335.401,A -85,B 0,C 180,E1 -6583.365,E2 -6583.365} C_VEL
LIN {X 0,Y 490.68,Z 323.758,A -85,B 0,C 180,E1 -6583.934,E2 -6583.934} C_VEL
LIN {X 0,Y 490.751,Z 313.915,A -85,B 0,C 180,E1 -6584.302,E2 -6584.302} C_VEL
LIN {X 0,Y 488.661,Z 301.219,A -85,B 0,C 180,E1 -6584.691,E2 -6584.691} C_VEL
LIN {X 0,Y 488.381,Z 299.529,A -85,B 0,C 180,E1 -6584.746,E2 -6584.746} C_VEL
LIN {X 0,Y 488.621,Z 289.615,A -85,B 0,C 180,E1 -6587.955,E2 -6587.955} C_VEL
LIN {X 0,Y 488.861,Z 280.036,A -85,B 0,C 180,E1 -6591.064,E2 -6591.064} C_VEL
LIN {X 0,Y 489.093,Z 270.433,A -85,B 0,C 180,E1 -6594.176,E2 -6594.176} C_VEL
LIN {X 0,Y 489.444,Z 260.916,A -85,B 0,C 180,E1 -6597.355,E2 -6597.355} C_VEL
LIN {X 0,Y 489.736,Z 251.573,A -85,B 0,C 180,E1 -6600.567,E2 -6600.567} C_VEL
LIN {X 0,Y 490.09,Z 242.711,A -85,B 0,C 180,E1 -6603.723,E2 -6603.723} C_VEL
LIN {X 0,Y 490.217,Z 236.549,A -85,B 0,C 180,E1 -6606.001,E2 -6606.001} C_VEL
LIN {X 0,Y 489.168,Z 230.107,A -85,B 0,C 180,E1 -6608.614,E2 -6608.614} C_VEL
LIN {X 0,Y 488.711,Z 227.613,A -85,B 0,C 180,E1 -6609.721,E2 -6609.721} C_VEL
LIN {X 0,Y 488.713,Z 227.611,A -85,B 0,C 180,E1 -6612.827,E2 -6612.827} C_VEL
LIN {X 0,Y 488.693,Z 227.611,A -85,B 0,C 180,E1 -6615.978,E2 -6615.978} C_VEL
LIN {X 0,Y 488.679,Z 227.614,A -85,B 0,C 180,E1 -6618.581,E2 -6618.581} C_VEL
LIN {X 0,Y 488.7,Z 227.61,A -85,B 0,C 180,E1 -6620.949,E2 -6620.949} C_VEL
LIN {X 0,Y 488.673,Z 227.614,A -85,B 0,C 180,E1 -6623.867,E2 -6623.867} C_VEL
LIN {X 0,Y 488.743,Z 227.606,A -85,B 0,C 180,E1 -6626.877,E2 -6626.877} C_VEL
LIN {X 0,Y 488.722,Z 227.607,A -85,B 0,C 180,E1 -6629.781,E2 -6629.781} C_VEL
LIN {X 0,Y 488.701,Z 227.608,A -85,B 0,C 180,E1 -6633.079,E2 -6633.079} C_VEL
LIN {X 0,Y 488.674,Z 227.615,A -85,B 0,C 180,E1 -6636.253,E2 -6636.253} C_VEL
LIN {X 0,Y 488.751,Z 227.604,A -85,B 0,C 180,E1 -6639.176,E2 -6639.176} C_VEL
LIN {X 0,Y 488.754,Z 227.604,A -85,B 0,C 180,E1 -6641.632,E2 -6641.632} C_VEL
LIN {X 0,Y 488.761,Z 227.602,A -85,B 0,C 180,E1 -6645,E2 -6645} C_VEL
LIN {X 0,Y 488.788,Z 227.598,A -85,B 0,C 180,E1 -6648.387,E2 -6648.387} C_VEL
LIN {X 0,Y 488.783,Z 227.601,A -85,B 0,C 180,E1 -6651.733,E2 -6651.733} C_VEL
LIN {X 0,Y 488.852,Z 227.592,A -85,B 0,C 180,E1 -6654.224,E2 -6654.224} C_VEL
LIN {X 0,Y 488.966,Z 227.577,A -85,B 0,C 180,E1 -6657.529,E2 -6657.529} C_VEL
LIN {X 0,Y 488.945,Z 227.581,A -85,B 0,C 180,E1 -6660,E2 -6660} C_VEL
LIN {X 0,Y 488.951,Z 227.576,A -85,B 0,C 180,E1 -6662.471,E2 -6662.471} C_VEL
LIN {X 0,Y 488.848,Z 227.591,A -85,B 0,C 180,E1 -6665.776,E2 -6665.776} C_VEL
LIN {X 0,Y 488.79,Z 227.6,A -85,B 0,C 180,E1 -6668.267,E2 -6668.267} C_VEL
LIN {X 0,Y 488.811,Z 227.599,A -85,B 0,C 180,E1 -6671.612,E2 -6671.612} C_VEL
LIN {X 0,Y 488.757,Z 227.605,A -85,B 0,C 180,E1 -6675.001,E2 -6675.001} C_VEL
LIN {X 0,Y 488.749,Z 227.604,A -85,B 0,C 180,E1 -6678.442,E2 -6678.442} C_VEL
LIN {X 0,Y 488.712,Z 227.608,A -85,B 0,C 180,E1 -6681.071,E2 -6681.071} C_VEL
LIN {X 0,Y 488.684,Z 227.613,A -85,B 0,C 180,E1 -6683.746,E2 -6683.746} C_VEL
LIN {X 0,Y 488.728,Z 227.607,A -85,B 0,C 180,E1 -6686.474,E2 -6686.474} C_VEL
LIN {X 0,Y 488.695,Z 227.61,A -85,B 0,C 180,E1 -6689.272,E2 -6689.272} C_VEL
LIN {X 0,Y 488.706,Z 227.61,A -85,B 0,C 180,E1 -6692.147,E2 -6692.147} C_VEL
LIN {X 0,Y 488.719,Z 227.607,A -85,B 0,C 180,E1 -6695.115,E2 -6695.115} C_VEL
LIN {X 0,Y 488.684,Z 227.612,A -85,B 0,C 180,E1 -6698.2,E2 -6698.2} C_VEL
LIN {X 0,Y 488.723,Z 227.608,A -85,B 0,C 180,E1 -6700.345,E2 -6700.345} C_VEL
LIN {X 0,Y 488.68,Z 227.612,A -85,B 0,C 180,E1 -6703.655,E2 -6703.655} C_VEL
LIN {X 0,Y 488.68,Z 227.613,A -85,B 0,C 180,E1 -6706.344,E2 -6706.344} C_VEL
LIN {X 0,Y 488.707,Z 227.613,A -85,B 0,C 180,E1 -6709.673,E2 -6709.673} C_VEL
LIN {X 0,Y 488.67,Z 227.615,A -85,B 0,C 180,E1 -6712.84,E2 -6712.84} C_VEL
LIN {X 0,Y 488.587,Z 227.626,A -85,B 0,C 180,E1 -6715.076,E2 -6715.076} C_VEL
LIN {X 0,Y 488.412,Z 227.649,A -85,B 0,C 180,E1 -6716.852,E2 -6716.852} C_VEL
LIN {X 0,Y 488.302,Z 229.216,A -85,B 0,C 180,E1 -6718.792,E2 -6718.792} C_VEL
LIN {X 0,Y 488.306,Z 232.095,A -85,B 0,C 180,E1 -6721.643,E2 -6721.643} C_VEL
LIN {X 0,Y 488.187,Z 234.785,A -85,B 0,C 180,E1 -6724.253,E2 -6724.253} C_VEL
LIN {X 0,Y 487.526,Z 235.563,A -85,B 0,C 180,E1 -6724.935,E2 -6724.935} C_VEL
LIN {X 0,Y 484.648,Z 236.979,A -85,B 0,C 180,E1 -6726.04,E2 -6726.04} C_VEL
LIN {X 0,Y 482.194,Z 238.121,A -85,B 0,C 180,E1 -6726.931,E2 -6726.931} C_VEL
LIN {X 0,Y 481.124,Z 238.93,A -85,B 0,C 180,E1 -6727.62,E2 -6727.62} C_VEL
LIN {X 0,Y 481.028,Z 239.181,A -85,B 0,C 180,E1 -6727.854,E2 -6727.854} C_VEL
LIN {X 0,Y 481.009,Z 241.889,A -85,B 0,C 180,E1 -6730.363,E2 -6730.363} C_VEL
LIN {X 0,Y 480.987,Z 244.887,A -85,B 0,C 180,E1 -6733.008,E2 -6733.008} C_VEL
LIN {X 0,Y 481.048,Z 247.603,A -85,B 0,C 180,E1 -6735.159,E2 -6735.159} C_VEL
LIN {X 0,Y 483.964,Z 260.514,A -85,B 0,C 180,E1 -6735.627,E2 -6735.627} C_VEL
LIN {X 0,Y 483.922,Z 272.549,A -85,B 0,C 180,E1 -6736.135,E2 -6736.135} C_VEL
LIN {X 0,Y 483.562,Z 284.148,A -85,B 0,C 180,E1 -6736.783,E2 -6736.783} C_VEL
LIN {X 0,Y 483.116,Z 295.549,A -85,B 0,C 180,E1 -6737.609,E2 -6737.609} C_VEL
LIN {X 0,Y 482.67,Z 305.982,A -85,B 0,C 180,E1 -6738.557,E2 -6738.557} C_VEL
LIN {X 0,Y 482.313,Z 314.501,A -85,B 0,C 180,E1 -6739.505,E2 -6739.505} C_VEL
LIN {X 0,Y 481.973,Z 322.342,A -85,B 0,C 180,E1 -6740.558,E2 -6740.558} C_VEL
LIN {X 0,Y 481.586,Z 330.009,A -85,B 0,C 180,E1 -6741.82,E2 -6741.82} C_VEL
LIN {X 0,Y 481.33,Z 337.031,A -85,B 0,C 180,E1 -6743.292,E2 -6743.292} C_VEL
LIN {X 0,Y 481.061,Z 341.715,A -85,B 0,C 180,E1 -6744.551,E2 -6744.551} C_VEL
LIN {X 0,Y 481.073,Z 345.289,A -85,B 0,C 180,E1 -6745.811,E2 -6745.811} C_VEL
LIN {X 0,Y 481.039,Z 347.138,A -85,B 0,C 180,E1 -6746.65,E2 -6746.65} C_VEL
LIN {X 0,Y 480.948,Z 348.537,A -85,B 0,C 180,E1 -6747.487,E2 -6747.487} C_VEL
LIN {X 0,Y 480.777,Z 350.147,A -85,B 0,C 180,E1 -6749.162,E2 -6749.162} C_VEL
LIN {X 0,Y 480.767,Z 350.382,A -85,B 0,C 180,E1 -6750,E2 -6750} C_VEL
LIN {X 0,Y 480.776,Z 350.198,A -85,B 0,C 180,E1 -6750.837,E2 -6750.837} C_VEL
LIN {X 0,Y 480.948,Z 348.653,A -85,B 0,C 180,E1 -6752.512,E2 -6752.512} C_VEL
LIN {X 0,Y 481.039,Z 347.306,A -85,B 0,C 180,E1 -6753.35,E2 -6753.35} C_VEL
LIN {X 0,Y 481.081,Z 344.465,A -85,B 0,C 180,E1 -6754.608,E2 -6754.608} C_VEL
LIN {X 0,Y 481.159,Z 340.61,A -85,B 0,C 180,E1 -6755.868,E2 -6755.868} C_VEL
LIN {X 0,Y 481.347,Z 335.633,A -85,B 0,C 180,E1 -6757.129,E2 -6757.129} C_VEL
LIN {X 0,Y 481.621,Z 329.36,A -85,B 0,C 180,E1 -6758.391,E2 -6758.391} C_VEL
LIN {X 0,Y 481.947,Z 321.505,A -85,B 0,C 180,E1 -6759.654,E2 -6759.654} C_VEL
LIN {X 0,Y 482.467,Z 311.721,A -85,B 0,C 180,E1 -6760.916,E2 -6760.916} C_VEL
LIN {X 0,Y 482.855,Z 301.459,A -85,B 0,C 180,E1 -6761.971,E2 -6761.971} C_VEL
LIN {X 0,Y 483.304,Z 290.521,A -85,B 0,C 180,E1 -6762.87,E2 -6762.87} C_VEL
LIN {X 0,Y 483.664,Z 280.144,A -85,B 0,C 180,E1 -6763.551,E2 -6763.551} C_VEL
LIN {X 0,Y 484.028,Z 267.615,A -85,B 0,C 180,E1 -6764.183,E2 -6764.183} C_VEL
LIN {X 0,Y 483.975,Z 260.439,A -85,B 0,C 180,E1 -6764.466,E2 -6764.466} C_VEL
LIN {X 0,Y 481.055,Z 247.424,A -85,B 0,C 180,E1 -6764.948,E2 -6764.948} C_VEL
LIN {X 0,Y 481.028,Z 243.551,A -85,B 0,C 180,E1 -6768.254,E2 -6768.254} C_VEL
LIN {X 0,Y 481.019,Z 240.039,A -85,B 0,C 180,E1 -6771.424,E2 -6771.424} C_VEL
LIN {X 0,Y 481.083,Z 237.194,A -85,B 0,C 180,E1 -6774.145,E2 -6774.145} C_VEL
LIN {X 0,Y 481.171,Z 234.256,A -85,B 0,C 180,E1 -6777.004,E2 -6777.004} C_VEL
LIN {X 0,Y 481.219,Z 231.482,A -85,B 0,C 180,E1 -6779.772,E2 -6779.772} C_VEL
LIN {X 0,Y 481.286,Z 228.559,A -85,B 0,C 180,E1 -6782.704,E2 -6782.704} C_VEL
LIN {X 0,Y 481.579,Z 228.499,A -85,B 0,C 180,E1 -6785.715,E2 -6785.715} C_VEL
LIN {X 0,Y 481.673,Z 228.487,A -85,B 0,C 180,E1 -6788.859,E2 -6788.859} C_VEL
LIN {X 0,Y 481.649,Z 228.489,A -85,B 0,C 180,E1 -6791.912,E2 -6791.912} C_VEL
LIN {X 0,Y 481.656,Z 228.487,A -85,B 0,C 180,E1 -6794.458,E2 -6794.458} C_VEL
LIN {X 0,Y 481.644,Z 228.491,A -85,B 0,C 180,E1 -6797.839,E2 -6797.839} C_VEL
LIN {X 0,Y 481.66,Z 228.488,A -85,B 0,C 180,E1 -6800.654,E2 -6800.654} C_VEL
LIN {X 0,Y 481.63,Z 228.491,A -85,B 0,C 180,E1 -6803.376,E2 -6803.376} C_VEL
LIN {X 0,Y 481.68,Z 228.484,A -85,B 0,C 180,E1 -6806.327,E2 -6806.327} C_VEL
LIN {X 0,Y 481.648,Z 228.492,A -85,B 0,C 180,E1 -6809.419,E2 -6809.419} C_VEL
LIN {X 0,Y 481.66,Z 228.487,A -85,B 0,C 180,E1 -6812.165,E2 -6812.165} C_VEL
LIN {X 0,Y 481.691,Z 228.485,A -85,B 0,C 180,E1 -6814.968,E2 -6814.968} C_VEL
LIN {X 0,Y 481.653,Z 228.491,A -85,B 0,C 180,E1 -6817.705,E2 -6817.705} C_VEL
LIN {X 0,Y 481.703,Z 228.481,A -85,B 0,C 180,E1 -6820.393,E2 -6820.393} C_VEL
LIN {X 0,Y 481.663,Z 228.49,A -85,B 0,C 180,E1 -6823.033,E2 -6823.033} C_VEL
LIN {X 0,Y 481.679,Z 228.484,A -85,B 0,C 180,E1 -6825.638,E2 -6825.638} C_VEL
LIN {X 0,Y 481.755,Z 228.476,A -85,B 0,C 180,E1 -6828.215,E2 -6828.215} C_VEL
LIN {X 0,Y 481.765,Z 228.475,A -85,B 0,C 180,E1 -6831.612,E2 -6831.612} C_VEL
LIN {X 0,Y 481.808,Z 228.468,A -85,B 0,C 180,E1 -6834.139,E2 -6834.139} C_VEL
LIN {X 0,Y 481.917,Z 228.452,A -85,B 0,C 180,E1 -6837.492,E2 -6837.492} C_VEL
LIN {X 0,Y 481.869,Z 228.461,A -85,B 0,C 180,E1 -6840.836,E2 -6840.836} C_VEL
LIN {X 0,Y 481.931,Z 228.454,A -85,B 0,C 180,E1 -6842.507,E2 -6842.507} C_VEL
LIN {X 0,Y 481.811,Z 228.469,A -85,B 0,C 180,E1 -6845.86,E2 -6845.86} C_VEL
LIN {X 0,Y 481.74,Z 228.479,A -85,B 0,C 180,E1 -6848.389,E2 -6848.389} C_VEL
LIN {X 0,Y 481.737,Z 228.477,A -85,B 0,C 180,E1 -6851.785,E2 -6851.785} C_VEL
LIN {X 0,Y 481.742,Z 228.477,A -85,B 0,C 180,E1 -6855.224,E2 -6855.224} C_VEL
LIN {X 0,Y 481.715,Z 228.481,A -85,B 0,C 180,E1 -6858.722,E2 -6858.722} C_VEL
LIN {X 0,Y 481.648,Z 228.488,A -85,B 0,C 180,E1 -6861.395,E2 -6861.395} C_VEL
LIN {X 0,Y 481.65,Z 228.491,A -85,B 0,C 180,E1 -6864.115,E2 -6864.115} C_VEL
LIN {X 0,Y 481.654,Z 228.487,A -85,B 0,C 180,E1 -6867.117,E2 -6867.117} C_VEL
LIN {X 0,Y 481.668,Z 228.487,A -85,B 0,C 180,E1 -6869.742,E2 -6869.742} C_VEL
LIN {X 0,Y 481.674,Z 228.486,A -85,B 0,C 180,E1 -6872.674,E2 -6872.674} C_VEL
LIN {X 0,Y 481.663,Z 228.487,A -85,B 0,C 180,E1 -6875.204,E2 -6875.204} C_VEL
LIN {X 0,Y 481.667,Z 228.485,A -85,B 0,C 180,E1 -6878.86,E2 -6878.86} C_VEL
LIN {X 0,Y 481.631,Z 228.489,A -85,B 0,C 180,E1 -6882.163,E2 -6882.163} C_VEL
LIN {X 0,Y 481.657,Z 228.488,A -85,B 0,C 180,E1 -6885.542,E2 -6885.542} C_VEL
LIN {X 0,Y 481.658,Z 228.49,A -85,B 0,C 180,E1 -6888.958,E2 -6888.958} C_VEL
LIN {X 0,Y 481.7,Z 228.553,A -85,B 0,C 180,E1 -6890.062,E2 -6890.062} C_VEL
LIN {X 0,Y 482.976,Z 235.864,A -85,B 0,C 180,E1 -6893.162,E2 -6893.162} C_VEL
LIN {X 0,Y 483.24,Z 239.354,A -85,B 0,C 180,E1 -6894.532,E2 -6894.532} C_VEL
LIN {X 0,Y 483.019,Z 245.804,A -85,B 0,C 180,E1 -6896.932,E2 -6896.932} C_VEL
LIN {X 0,Y 482.658,Z 253.916,A -85,B 0,C 180,E1 -6899.844,E2 -6899.844} C_VEL
LIN {X 0,Y 482.329,Z 263.42,A -85,B 0,C 180,E1 -6903.147,E2 -6903.147} C_VEL
LIN {X 0,Y 482.003,Z 272.937,A -85,B 0,C 180,E1 -6906.361,E2 -6906.361} C_VEL
LIN {X 0,Y 481.772,Z 282.503,A -85,B 0,C 180,E1 -6909.506,E2 -6909.506} C_VEL
LIN {X 0,Y 481.503,Z 292.077,A -85,B 0,C 180,E1 -6912.589,E2 -6912.589} C_VEL
LIN {X 0,Y 481.332,Z 299.582,A -85,B 0,C 180,E1 -6915.05,E2 -6915.05} C_VEL
LIN {X 0,Y 483.613,Z 313.096,A -85,B 0,C 180,E1 -6915.455,E2 -6915.455} C_VEL
LIN {X 0,Y 483.964,Z 317.741,A -85,B 0,C 180,E1 -6915.627,E2 -6915.627} C_VEL
LIN {X 0,Y 483.561,Z 330.51,A -85,B 0,C 180,E1 -6916.178,E2 -6916.178} C_VEL
LIN {X 0,Y 483.089,Z 342.678,A -85,B 0,C 180,E1 -6916.893,E2 -6916.893} C_VEL
LIN {X 0,Y 482.698,Z 353.485,A -85,B 0,C 180,E1 -6917.705,E2 -6917.705} C_VEL
LIN {X 0,Y 482.302,Z 363.646,A -85,B 0,C 180,E1 -6918.655,E2 -6918.655} C_VEL
LIN {X 0,Y 481.882,Z 372.786,A -85,B 0,C 180,E1 -6919.708,E2 -6919.708} C_VEL
LIN {X 0,Y 481.531,Z 381.688,A -85,B 0,C 180,E1 -6920.973,E2 -6920.973} C_VEL
LIN {X 0,Y 481.207,Z 388.849,A -85,B 0,C 180,E1 -6922.236,E2 -6922.236} C_VEL
LIN {X 0,Y 481.048,Z 394.357,A -85,B 0,C 180,E1 -6923.448,E2 -6923.448} C_VEL
LIN {X 0,Y 480.998,Z 398.373,A -85,B 0,C 180,E1 -6924.55,E2 -6924.55} C_VEL
LIN {X 0,Y 480.847,Z 401.958,A -85,B 0,C 180,E1 -6925.809,E2 -6925.809} C_VEL
LIN {X 0,Y 480.891,Z 403.807,A -85,B 0,C 180,E1 -6926.649,E2 -6926.649} C_VEL
LIN {X 0,Y 480.79,Z 406.182,A -85,B 0,C 180,E1 -6928.325,E2 -6928.325} C_VEL
LIN {X 0,Y 480.743,Z 407,A -85,B 0,C 180,E1 -6930,E2 -6930} C_VEL
LIN {X 0,Y 480.79,Z 406.184,A -85,B 0,C 180,E1 -6931.675,E2 -6931.675} C_VEL
LIN {X 0,Y 480.891,Z 403.81,A -85,B 0,C 180,E1 -6933.351,E2 -6933.351} C_VEL
LIN {X 0,Y 480.854,Z 400.895,A -85,B 0,C 180,E1 -6934.611,E2 -6934.611} C_VEL
LIN {X 0,Y 481.023,Z 396.948,A -85,B 0,C 180,E1 -6935.87,E2 -6935.87} C_VEL
LIN {X 0,Y 481.116,Z 390.875,A -85,B 0,C 180,E1 -6937.344,E2 -6937.344} C_VEL
LIN {X 0,Y 481.426,Z 384.234,A -85,B 0,C 180,E1 -6938.606,E2 -6938.606} C_VEL
LIN {X 0,Y 481.756,Z 375.99,A -85,B 0,C 180,E1 -6939.87,E2 -6939.87} C_VEL
LIN {X 0,Y 482.108,Z 367.538,A -85,B 0,C 180,E1 -6940.924,E2 -6940.924} C_VEL
LIN {X 0,Y 482.565,Z 357.089,A -85,B 0,C 180,E1 -6941.978,E2 -6941.978} C_VEL
LIN {X 0,Y 482.967,Z 345.875,A -85,B 0,C 180,E1 -6942.887,E2 -6942.887} C_VEL
LIN {X 0,Y 483.367,Z 335.401,A -85,B 0,C 180,E1 -6943.56,E2 -6943.56} C_VEL
LIN {X 0,Y 483.8,Z 323.758,A -85,B 0,C 180,E1 -6944.137,E2 -6944.137} C_VEL
LIN {X 0,Y 483.825,Z 314.678,A -85,B 0,C 180,E1 -6944.485,E2 -6944.485} C_VEL
LIN {X 0,Y 481.702,Z 301.594,A -85,B 0,C 180,E1 -6944.901,E2 -6944.901} C_VEL
LIN {X 0,Y 481.323,Z 299.529,A -85,B 0,C 180,E1 -6944.967,E2 -6944.967} C_VEL
LIN {X 0,Y 481.556,Z 290.71,A -85,B 0,C 180,E1 -6947.848,E2 -6947.848} C_VEL
LIN {X 0,Y 481.797,Z 280.93,A -85,B 0,C 180,E1 -6951.001,E2 -6951.001} C_VEL
LIN {X 0,Y 482.028,Z 271.541,A -85,B 0,C 180,E1 -6954.095,E2 -6954.095} C_VEL
LIN {X 0,Y 482.401,Z 262.126,A -85,B 0,C 180,E1 -6957.29,E2 -6957.29} C_VEL
LIN {X 0,Y 482.746,Z 252.093,A -85,B 0,C 180,E1 -6960.801,E2 -6960.801} C_VEL
LIN {X 0,Y 483.133,Z 243.293,A -85,B 0,C 180,E1 -6963.987,E2 -6963.987} C_VEL
LIN {X 0,Y 483.243,Z 237.739,A -85,B 0,C 180,E1 -6966.087,E2 -6966.087} C_VEL
LIN {X 0,Y 482.16,Z 231.129,A -85,B 0,C 180,E1 -6968.813,E2 -6968.813} C_VEL
LIN {X 0,Y 481.684,Z 228.489,A -85,B 0,C 180,E1 -6970.005,E2 -6970.005} C_VEL
LIN {X 0,Y 481.642,Z 228.495,A -85,B 0,C 180,E1 -6973.3,E2 -6973.3} C_VEL
LIN {X 0,Y 481.656,Z 228.49,A -85,B 0,C 180,E1 -6975.642,E2 -6975.642} C_VEL
LIN {X 0,Y 481.634,Z 228.492,A -85,B 0,C 180,E1 -6978.956,E2 -6978.956} C_VEL
LIN {X 0,Y 481.651,Z 228.488,A -85,B 0,C 180,E1 -6981.994,E2 -6981.994} C_VEL
LIN {X 0,Y 481.692,Z 228.484,A -85,B 0,C 180,E1 -6985.318,E2 -6985.318} C_VEL
LIN {X 0,Y 481.648,Z 228.489,A -85,B 0,C 180,E1 -6988.312,E2 -6988.312} C_VEL
LIN {X 0,Y 481.663,Z 228.486,A -85,B 0,C 180,E1 -6991.216,E2 -6991.216} C_VEL
LIN {X 0,Y 481.646,Z 228.49,A -85,B 0,C 180,E1 -6994.04,E2 -6994.04} C_VEL
LIN {X 0,Y 481.678,Z 228.484,A -85,B 0,C 180,E1 -6996.812,E2 -6996.812} C_VEL
LIN {X 0,Y 481.7,Z 228.484,A -85,B 0,C 180,E1 -6999.503,E2 -6999.503} C_VEL
LIN {X 0,Y 481.697,Z 228.483,A -85,B 0,C 180,E1 -7002.158,E2 -7002.158} C_VEL
LIN {X 0,Y 481.744,Z 228.476,A -85,B 0,C 180,E1 -7004.776,E2 -7004.776} C_VEL
LIN {X 0,Y 481.739,Z 228.477,A -85,B 0,C 180,E1 -7008.215,E2 -7008.215} C_VEL
LIN {X 0,Y 481.736,Z 228.48,A -85,B 0,C 180,E1 -7011.611,E2 -7011.611} C_VEL
LIN {X 0,Y 481.813,Z 228.469,A -85,B 0,C 180,E1 -7014.14,E2 -7014.14} C_VEL
LIN {X 0,Y 481.932,Z 228.454,A -85,B 0,C 180,E1 -7017.493,E2 -7017.493} C_VEL
LIN {X 0,Y 481.915,Z 228.456,A -85,B 0,C 180,E1 -7020,E2 -7020} C_VEL
LIN {X 0,Y 481.918,Z 228.452,A -85,B 0,C 180,E1 -7022.508,E2 -7022.508} C_VEL
LIN {X 0,Y 481.809,Z 228.468,A -85,B 0,C 180,E1 -7025.861,E2 -7025.861} C_VEL
LIN {X 0,Y 481.745,Z 228.477,A -85,B 0,C 180,E1 -7028.389,E2 -7028.389} C_VEL
LIN {X 0,Y 481.756,Z 228.476,A -85,B 0,C 180,E1 -7031.785,E2 -7031.785} C_VEL
LIN {X 0,Y 481.742,Z 228.48,A -85,B 0,C 180,E1 -7035.224,E2 -7035.224} C_VEL
LIN {X 0,Y 481.711,Z 228.484,A -85,B 0,C 180,E1 -7038.722,E2 -7038.722} C_VEL
LIN {X 0,Y 481.651,Z 228.488,A -85,B 0,C 180,E1 -7041.395,E2 -7041.395} C_VEL
LIN {X 0,Y 481.666,Z 228.488,A -85,B 0,C 180,E1 -7044.114,E2 -7044.114} C_VEL
LIN {X 0,Y 481.698,Z 228.484,A -85,B 0,C 180,E1 -7047.127,E2 -7047.127} C_VEL
LIN {X 0,Y 481.66,Z 228.485,A -85,B 0,C 180,E1 -7049.743,E2 -7049.743} C_VEL
LIN {X 0,Y 481.674,Z 228.486,A -85,B 0,C 180,E1 -7052.674,E2 -7052.674} C_VEL
LIN {X 0,Y 481.64,Z 228.49,A -85,B 0,C 180,E1 -7055.709,E2 -7055.709} C_VEL
LIN {X 0,Y 481.675,Z 228.487,A -85,B 0,C 180,E1 -7058.859,E2 -7058.859} C_VEL
LIN {X 0,Y 481.65,Z 228.488,A -85,B 0,C 180,E1 -7061.912,E2 -7061.912} C_VEL
LIN {X 0,Y 481.657,Z 228.489,A -85,B 0,C 180,E1 -7064.458,E2 -7064.458} C_VEL
LIN {X 0,Y 481.646,Z 228.493,A -85,B 0,C 180,E1 -7067.839,E2 -7067.839} C_VEL
LIN {X 0,Y 481.664,Z 228.487,A -85,B 0,C 180,E1 -7070.654,E2 -7070.654} C_VEL
LIN {X 0,Y 481.617,Z 228.494,A -85,B 0,C 180,E1 -7073.378,E2 -7073.378} C_VEL
LIN {X 0,Y 481.413,Z 228.52,A -85,B 0,C 180,E1 -7076.318,E2 -7076.318} C_VEL
LIN {X 0,Y 481.292,Z 228.536,A -85,B 0,C 180,E1 -7077.296,E2 -7077.296} C_VEL
LIN {X 0,Y 481.221,Z 231.392,A -85,B 0,C 180,E1 -7080.227,E2 -7080.227} C_VEL
LIN {X 0,Y 481.167,Z 234.271,A -85,B 0,C 180,E1 -7083.077,E2 -7083.077} C_VEL
LIN {X 0,Y 481.088,Z 237.108,A -85,B 0,C 180,E1 -7085.855,E2 -7085.855} C_VEL
LIN {X 0,Y 481.028,Z 239.181,A -85,B 0,C 180,E1 -7087.854,E2 -7087.854} C_VEL
LIN {X 0,Y 480.332,Z 239.979,A -85,B 0,C 180,E1 -7088.546,E2 -7088.546} C_VEL
LIN {X 0,Y 477.449,Z 241.471,A -85,B 0,C 180,E1 -7089.667,E2 -7089.667} C_VEL
LIN {X 0,Y 475.04,Z 242.697,A -85,B 0,C 180,E1 -7090.57,E2 -7090.57} C_VEL
LIN {X 0,Y 474.027,Z 243.573,A -85,B 0,C 180,E1 -7091.269,E2 -7091.269} C_VEL
LIN {X 0,Y 473.956,Z 243.846,A -85,B 0,C 180,E1 -7091.506,E2 -7091.506} C_VEL
LIN {X 0,Y 473.99,Z 247.892,A -85,B 0,C 180,E1 -7094.926,E2 -7094.926} C_VEL
LIN {X 0,Y 477.124,Z 261.722,A -85,B 0,C 180,E1 -7095.444,E2 -7095.444} C_VEL
LIN {X 0,Y 477.053,Z 272.986,A -85,B 0,C 180,E1 -7095.931,E2 -7095.931} C_VEL
LIN {X 0,Y 476.685,Z 284.497,A -85,B 0,C 180,E1 -7096.583,E2 -7096.583} C_VEL
LIN {X 0,Y 476.216,Z 295.98,A -85,B 0,C 180,E1 -7097.427,E2 -7097.427} C_VEL
LIN {X 0,Y 475.729,Z 306.414,A -85,B 0,C 180,E1 -7098.388,E2 -7098.388} C_VEL
LIN {X 0,Y 475.357,Z 314.931,A -85,B 0,C 180,E1 -7099.35,E2 -7099.35} C_VEL
LIN {X 0,Y 474.989,Z 322.772,A -85,B 0,C 180,E1 -7100.418,E2 -7100.418} C_VEL
LIN {X 0,Y 474.577,Z 330.438,A -85,B 0,C 180,E1 -7101.698,E2 -7101.698} C_VEL
LIN {X 0,Y 474.268,Z 337.461,A -85,B 0,C 180,E1 -7103.191,E2 -7103.191} C_VEL
LIN {X 0,Y 474.009,Z 342.144,A -85,B 0,C 180,E1 -7104.469,E2 -7104.469} C_VEL
LIN {X 0,Y 474.021,Z 345.716,A -85,B 0,C 180,E1 -7105.749,E2 -7105.749} C_VEL
LIN {X 0,Y 473.963,Z 347.566,A -85,B 0,C 180,E1 -7106.599,E2 -7106.599} C_VEL
LIN {X 0,Y 473.891,Z 348.963,A -85,B 0,C 180,E1 -7107.45,E2 -7107.45} C_VEL
LIN {X 0,Y 473.704,Z 350.574,A -85,B 0,C 180,E1 -7109.15,E2 -7109.15} C_VEL
LIN {X 0,Y 473.692,Z 350.808,A -85,B 0,C 180,E1 -7110,E2 -7110} C_VEL
LIN {X 0,Y 473.704,Z 350.624,A -85,B 0,C 180,E1 -7110.85,E2 -7110.85} C_VEL
LIN {X 0,Y 473.891,Z 349.078,A -85,B 0,C 180,E1 -7112.55,E2 -7112.55} C_VEL
LIN {X 0,Y 473.963,Z 347.732,A -85,B 0,C 180,E1 -7113.4,E2 -7113.4} C_VEL
LIN {X 0,Y 474.022,Z 344.89,A -85,B 0,C 180,E1 -7114.677,E2 -7114.677} C_VEL
LIN {X 0,Y 474.12,Z 341.035,A -85,B 0,C 180,E1 -7115.956,E2 -7115.956} C_VEL
LIN {X 0,Y 474.308,Z 336.056,A -85,B 0,C 180,E1 -7117.235,E2 -7117.235} C_VEL
LIN {X 0,Y 474.62,Z 329.783,A -85,B 0,C 180,E1 -7118.515,E2 -7118.515} C_VEL
LIN {X 0,Y 474.951,Z 321.929,A -85,B 0,C 180,E1 -7119.798,E2 -7119.798} C_VEL
LIN {X 0,Y 475.498,Z 312.145,A -85,B 0,C 180,E1 -7121.078,E2 -7121.078} C_VEL
LIN {X 0,Y 475.941,Z 301.879,A -85,B 0,C 180,E1 -7122.147,E2 -7122.147} C_VEL
LIN {X 0,Y 476.379,Z 291.487,A -85,B 0,C 180,E1 -7123.018,E2 -7123.018} C_VEL
LIN {X 0,Y 476.795,Z 280.562,A -85,B 0,C 180,E1 -7123.75,E2 -7123.75} C_VEL
LIN {X 0,Y 477.166,Z 268.03,A -85,B 0,C 180,E1 -7124.391,E2 -7124.391} C_VEL
LIN {X 0,Y 477.149,Z 261.63,A -85,B 0,C 180,E1 -7124.65,E2 -7124.65} C_VEL
LIN {X 0,Y 474.068,Z 248.557,A -85,B 0,C 180,E1 -7125.144,E2 -7125.144} C_VEL
LIN {X 0,Y 473.976,Z 247.795,A -85,B 0,C 180,E1 -7125.201,E2 -7125.201} C_VEL
LIN {X 0,Y 473.963,Z 244.094,A -85,B 0,C 180,E1 -7128.376,E2 -7128.376} C_VEL
LIN {X 0,Y 473.944,Z 240.368,A -85,B 0,C 180,E1 -7131.76,E2 -7131.76} C_VEL
LIN {X 0,Y 474.03,Z 237.502,A -85,B 0,C 180,E1 -7134.528,E2 -7134.528} C_VEL
LIN {X 0,Y 474.102,Z 234.614,A -85,B 0,C 180,E1 -7137.357,E2 -7137.357} C_VEL
LIN {X 0,Y 474.157,Z 231.727,A -85,B 0,C 180,E1 -7140.262,E2 -7140.262} C_VEL
LIN {X 0,Y 474.22,Z 229.649,A -85,B 0,C 180,E1 -7142.355,E2 -7142.355} C_VEL
LIN {X 0,Y 474.396,Z 229.396,A -85,B 0,C 180,E1 -7144.261,E2 -7144.261} C_VEL
LIN {X 0,Y 474.562,Z 229.373,A -85,B 0,C 180,E1 -7146.897,E2 -7146.897} C_VEL
LIN {X 0,Y 474.616,Z 229.365,A -85,B 0,C 180,E1 -7149.645,E2 -7149.645} C_VEL
LIN {X 0,Y 474.602,Z 229.37,A -85,B 0,C 180,E1 -7152.233,E2 -7152.233} C_VEL
LIN {X 0,Y 474.618,Z 229.363,A -85,B 0,C 180,E1 -7155.298,E2 -7155.298} C_VEL
LIN {X 0,Y 474.616,Z 229.364,A -85,B 0,C 180,E1 -7158.214,E2 -7158.214} C_VEL
LIN {X 0,Y 474.614,Z 229.366,A -85,B 0,C 180,E1 -7161.543,E2 -7161.543} C_VEL
LIN {X 0,Y 474.625,Z 229.363,A -85,B 0,C 180,E1 -7164.726,E2 -7164.726} C_VEL
LIN {X 0,Y 474.637,Z 229.364,A -85,B 0,C 180,E1 -7167.788,E2 -7167.788} C_VEL
LIN {X 0,Y 474.601,Z 229.366,A -85,B 0,C 180,E1 -7170.89,E2 -7170.89} C_VEL
LIN {X 0,Y 474.618,Z 229.365,A -85,B 0,C 180,E1 -7173.626,E2 -7173.626} C_VEL
LIN {X 0,Y 474.637,Z 229.363,A -85,B 0,C 180,E1 -7176.642,E2 -7176.642} C_VEL
LIN {X 0,Y 474.655,Z 229.359,A -85,B 0,C 180,E1 -7180.089,E2 -7180.089} C_VEL
LIN {X 0,Y 474.626,Z 229.363,A -85,B 0,C 180,E1 -7182.773,E2 -7182.773} C_VEL
LIN {X 0,Y 474.639,Z 229.361,A -85,B 0,C 180,E1 -7185.421,E2 -7185.421} C_VEL
LIN {X 0,Y 474.708,Z 229.353,A -85,B 0,C 180,E1 -7188.038,E2 -7188.038} C_VEL
LIN {X 0,Y 474.731,Z 229.352,A -85,B 0,C 180,E1 -7191.486,E2 -7191.486} C_VEL
LIN {X 0,Y 474.771,Z 229.345,A -85,B 0,C 180,E1 -7194.052,E2 -7194.052} C_VEL
LIN {X 0,Y 474.883,Z 229.329,A -85,B 0,C 180,E1 -7197.455,E2 -7197.455} C_VEL
LIN {X 0,Y 474.882,Z 229.332,A -85,B 0,C 180,E1 -7200,E2 -7200} C_VEL
LIN {X 0,Y 474.897,Z 229.33,A -85,B 0,C 180,E1 -7202.545,E2 -7202.545} C_VEL
LIN {X 0,Y 474.774,Z 229.345,A -85,B 0,C 180,E1 -7205.948,E2 -7205.948} C_VEL
LIN {X 0,Y 474.711,Z 229.356,A -85,B 0,C 180,E1 -7208.514,E2 -7208.514} C_VEL
LIN {X 0,Y 474.695,Z 229.356,A -85,B 0,C 180,E1 -7211.963,E2 -7211.963} C_VEL
LIN {X 0,Y 474.702,Z 229.354,A -85,B 0,C 180,E1 -7215.456,E2 -7215.456} C_VEL
LIN {X 0,Y 474.668,Z 229.359,A -85,B 0,C 180,E1 -7219.01,E2 -7219.01} C_VEL
LIN {X 0,Y 474.591,Z 229.368,A -85,B 0,C 180,E1 -7221.729,E2 -7221.729} C_VEL
LIN {X 0,Y 474.628,Z 229.362,A -85,B 0,C 180,E1 -7224.495,E2 -7224.495} C_VEL
LIN {X 0,Y 474.601,Z 229.367,A -85,B 0,C 180,E1 -7227.326,E2 -7227.326} C_VEL
LIN {X 0,Y 474.6,Z 229.367,A -85,B 0,C 180,E1 -7230.231,E2 -7230.231} C_VEL
LIN {X 0,Y 474.645,Z 229.362,A -85,B 0,C 180,E1 -7233.22,E2 -7233.22} C_VEL
LIN {X 0,Y 474.586,Z 229.368,A -85,B 0,C 180,E1 -7236.324,E2 -7236.324} C_VEL
LIN {X 0,Y 474.623,Z 229.367,A -85,B 0,C 180,E1 -7239.548,E2 -7239.548} C_VEL
LIN {X 0,Y 474.59,Z 229.367,A -85,B 0,C 180,E1 -7242.232,E2 -7242.232} C_VEL
LIN {X 0,Y 474.619,Z 229.365,A -85,B 0,C 180,E1 -7245.298,E2 -7245.298} C_VEL
LIN {X 0,Y 474.623,Z 229.366,A -85,B 0,C 180,E1 -7248.215,E2 -7248.215} C_VEL
LIN {X 0,Y 474.647,Z 229.365,A -85,B 0,C 180,E1 -7249.739,E2 -7249.739} C_VEL
LIN {X 0,Y 475.917,Z 236.632,A -85,B 0,C 180,E1 -7252.886,E2 -7252.886} C_VEL
LIN {X 0,Y 476.278,Z 240.018,A -85,B 0,C 180,E1 -7254.251,E2 -7254.251} C_VEL
LIN {X 0,Y 476.043,Z 246.966,A -85,B 0,C 180,E1 -7256.89,E2 -7256.89} C_VEL
LIN {X 0,Y 475.647,Z 255.078,A -85,B 0,C 180,E1 -7259.843,E2 -7259.843} C_VEL
LIN {X 0,Y 475.294,Z 264.557,A -85,B 0,C 180,E1 -7263.193,E2 -7263.193} C_VEL
LIN {X 0,Y 474.985,Z 272.696,A -85,B 0,C 180,E1 -7265.99,E2 -7265.99} C_VEL
LIN {X 0,Y 474.712,Z 282.225,A -85,B 0,C 180,E1 -7269.187,E2 -7269.187} C_VEL
LIN {X 0,Y 474.469,Z 291.788,A -85,B 0,C 180,E1 -7272.323,E2 -7272.323} C_VEL
LIN {X 0,Y 474.263,Z 299.6,A -85,B 0,C 180,E1 -7274.826,E2 -7274.826} C_VEL
LIN {X 0,Y 476.613,Z 313.096,A -85,B 0,C 180,E1 -7275.237,E2 -7275.237} C_VEL
LIN {X 0,Y 477.079,Z 318.503,A -85,B 0,C 180,E1 -7275.442,E2 -7275.442} C_VEL
LIN {X 0,Y 476.666,Z 330.51,A -85,B 0,C 180,E1 -7275.974,E2 -7275.974} C_VEL
LIN {X 0,Y 476.175,Z 342.677,A -85,B 0,C 180,E1 -7276.699,E2 -7276.699} C_VEL
LIN {X 0,Y 475.738,Z 353.734,A -85,B 0,C 180,E1 -7277.544,E2 -7277.544} C_VEL
LIN {X 0,Y 475.339,Z 363.646,A -85,B 0,C 180,E1 -7278.486,E2 -7278.486} C_VEL
LIN {X 0,Y 474.886,Z 372.786,A -85,B 0,C 180,E1 -7279.555,E2 -7279.555} C_VEL
LIN {X 0,Y 474.482,Z 381.688,A -85,B 0,C 180,E1 -7280.838,E2 -7280.838} C_VEL
LIN {X 0,Y 474.152,Z 388.849,A -85,B 0,C 180,E1 -7282.12,E2 -7282.12} C_VEL
LIN {X 0,Y 473.972,Z 394.739,A -85,B 0,C 180,E1 -7283.449,E2 -7283.449} C_VEL
LIN {X 0,Y 473.845,Z 399.677,A -85,B 0,C 180,E1 -7284.895,E2 -7284.895} C_VEL
LIN {X 0,Y 473.752,Z 401.958,A -85,B 0,C 180,E1 -7285.746,E2 -7285.746} C_VEL
LIN {X 0,Y 473.799,Z 403.807,A -85,B 0,C 180,E1 -7286.599,E2 -7286.599} C_VEL
LIN {X 0,Y 473.695,Z 406.182,A -85,B 0,C 180,E1 -7288.3,E2 -7288.3} C_VEL
LIN {X 0,Y 473.688,Z 406.786,A -85,B 0,C 180,E1 -7289.15,E2 -7289.15} C_VEL
LIN {X 0,Y 473.669,Z 407,A -85,B 0,C 180,E1 -7290,E2 -7290} C_VEL
LIN {X 0,Y 473.688,Z 406.786,A -85,B 0,C 180,E1 -7290.85,E2 -7290.85} C_VEL
LIN {X 0,Y 473.724,Z 405.196,A -85,B 0,C 180,E1 -7292.551,E2 -7292.551} C_VEL
LIN {X 0,Y 473.799,Z 403.81,A -85,B 0,C 180,E1 -7293.402,E2 -7293.402} C_VEL
LIN {X 0,Y 473.776,Z 400.895,A -85,B 0,C 180,E1 -7294.68,E2 -7294.68} C_VEL
LIN {X 0,Y 473.942,Z 396.947,A -85,B 0,C 180,E1 -7295.958,E2 -7295.958} C_VEL
LIN {X 0,Y 474.049,Z 390.875,A -85,B 0,C 180,E1 -7297.454,E2 -7297.454} C_VEL
LIN {X 0,Y 474.378,Z 384.234,A -85,B 0,C 180,E1 -7298.735,E2 -7298.735} C_VEL
LIN {X 0,Y 474.752,Z 375.991,A -85,B 0,C 180,E1 -7300.017,E2 -7300.017} C_VEL
LIN {X 0,Y 475.116,Z 367.538,A -85,B 0,C 180,E1 -7301.087,E2 -7301.087} C_VEL
LIN {X 0,Y 475.607,Z 357.106,A -85,B 0,C 180,E1 -7302.154,E2 -7302.154} C_VEL
LIN {X 0,Y 476.026,Z 346.037,A -85,B 0,C 180,E1 -7303.066,E2 -7303.066} C_VEL
LIN {X 0,Y 476.454,Z 335.4,A -85,B 0,C 180,E1 -7303.76,E2 -7303.76} C_VEL
LIN {X 0,Y 476.908,Z 323.758,A -85,B 0,C 180,E1 -7304.345,E2 -7304.345} C_VEL
LIN {X 0,Y 476.909,Z 315.438,A -85,B 0,C 180,E1 -7304.672,E2 -7304.672} C_VEL
LIN {X 0,Y 474.912,Z 302.986,A -85,B 0,C 180,E1 -7305.089,E2 -7305.089} C_VEL
LIN {X 0,Y 474.272,Z 299.433,A -85,B 0,C 180,E1 -7305.195,E2 -7305.195} C_VEL
LIN {X 0,Y 474.544,Z 288.946,A -85,B 0,C 180,E1 -7308.587,E2 -7308.587} C_VEL
LIN {X 0,Y 474.814,Z 279.447,A -85,B 0,C 180,E1 -7311.718,E2 -7311.718} C_VEL
LIN {X 0,Y 475.09,Z 269.903,A -85,B 0,C 180,E1 -7314.936,E2 -7314.936} C_VEL
LIN {X 0,Y 475.411,Z 261.643,A -85,B 0,C 180,E1 -7317.819,E2 -7317.819} C_VEL
LIN {X 0,Y 475.774,Z 252.363,A -85,B 0,C 180,E1 -7321.132,E2 -7321.132} C_VEL
LIN {X 0,Y 476.184,Z 243.889,A -85,B 0,C 180,E1 -7324.258,E2 -7324.258} C_VEL
LIN {X 0,Y 476.252,Z 238.913,A -85,B 0,C 180,E1 -7326.177,E2 -7326.177} C_VEL
LIN {X 0,Y 475.157,Z 232.311,A -85,B 0,C 180,E1 -7328.948,E2 -7328.948} C_VEL
LIN {X 0,Y 474.667,Z 229.363,A -85,B 0,C 180,E1 -7330.259,E2 -7330.259} C_VEL
LIN {X 0,Y 474.604,Z 229.372,A -85,B 0,C 180,E1 -7333.481,E2 -7333.481} C_VEL
LIN {X 0,Y 474.592,Z 229.367,A -85,B 0,C 180,E1 -7336.521,E2 -7336.521} C_VEL
LIN {X 0,Y 474.597,Z 229.365,A -85,B 0,C 180,E1 -7339.34,E2 -7339.34} C_VEL
LIN {X 0,Y 474.609,Z 229.364,A -85,B 0,C 180,E1 -7341.705,E2 -7341.705} C_VEL
LIN {X 0,Y 474.626,Z 229.364,A -85,B 0,C 180,E1 -7344.726,E2 -7344.726} C_VEL
LIN {X 0,Y 474.639,Z 229.363,A -85,B 0,C 180,E1 -7347.788,E2 -7347.788} C_VEL
LIN {X 0,Y 474.602,Z 229.367,A -85,B 0,C 180,E1 -7350.89,E2 -7350.89} C_VEL
LIN {X 0,Y 474.593,Z 229.365,A -85,B 0,C 180,E1 -7353.624,E2 -7353.624} C_VEL
LIN {X 0,Y 474.638,Z 229.361,A -85,B 0,C 180,E1 -7356.642,E2 -7356.642} C_VEL
LIN {X 0,Y 474.659,Z 229.36,A -85,B 0,C 180,E1 -7360.09,E2 -7360.09} C_VEL
LIN {X 0,Y 474.644,Z 229.362,A -85,B 0,C 180,E1 -7362.774,E2 -7362.774} C_VEL
LIN {X 0,Y 474.644,Z 229.36,A -85,B 0,C 180,E1 -7365.421,E2 -7365.421} C_VEL
LIN {X 0,Y 474.697,Z 229.356,A -85,B 0,C 180,E1 -7368.037,E2 -7368.037} C_VEL
LIN {X 0,Y 474.707,Z 229.357,A -85,B 0,C 180,E1 -7371.486,E2 -7371.486} C_VEL
LIN {X 0,Y 474.775,Z 229.345,A -85,B 0,C 180,E1 -7374.052,E2 -7374.052} C_VEL
LIN {X 0,Y 474.898,Z 229.33,A -85,B 0,C 180,E1 -7377.455,E2 -7377.455} C_VEL
LIN {X 0,Y 474.884,Z 229.332,A -85,B 0,C 180,E1 -7380,E2 -7380} C_VEL
LIN {X 0,Y 474.884,Z 229.328,A -85,B 0,C 180,E1 -7382.545,E2 -7382.545} C_VEL
LIN {X 0,Y 474.772,Z 229.344,A -85,B 0,C 180,E1 -7385.948,E2 -7385.948} C_VEL
LIN {X 0,Y 474.716,Z 229.353,A -85,B 0,C 180,E1 -7388.514,E2 -7388.514} C_VEL
LIN {X 0,Y 474.71,Z 229.353,A -85,B 0,C 180,E1 -7391.962,E2 -7391.962} C_VEL
LIN {X 0,Y 474.684,Z 229.354,A -85,B 0,C 180,E1 -7395.767,E2 -7395.767} C_VEL
LIN {X 0,Y 474.665,Z 229.36,A -85,B 0,C 180,E1 -7399.01,E2 -7399.01} C_VEL
LIN {X 0,Y 474.594,Z 229.367,A -85,B 0,C 180,E1 -7401.729,E2 -7401.729} C_VEL
LIN {X 0,Y 474.645,Z 229.362,A -85,B 0,C 180,E1 -7404.494,E2 -7404.494} C_VEL
LIN {X 0,Y 474.641,Z 229.362,A -85,B 0,C 180,E1 -7407.324,E2 -7407.324} C_VEL
LIN {X 0,Y 474.599,Z 229.368,A -85,B 0,C 180,E1 -7410.808,E2 -7410.808} C_VEL
LIN {X 0,Y 474.629,Z 229.361,A -85,B 0,C 180,E1 -7413.221,E2 -7413.221} C_VEL
LIN {X 0,Y 474.593,Z 229.368,A -85,B 0,C 180,E1 -7416.323,E2 -7416.323} C_VEL
LIN {X 0,Y 474.63,Z 229.364,A -85,B 0,C 180,E1 -7419.548,E2 -7419.548} C_VEL
LIN {X 0,Y 474.604,Z 229.368,A -85,B 0,C 180,E1 -7422.233,E2 -7422.233} C_VEL
LIN {X 0,Y 474.62,Z 229.362,A -85,B 0,C 180,E1 -7425.298,E2 -7425.298} C_VEL
LIN {X 0,Y 474.617,Z 229.365,A -85,B 0,C 180,E1 -7428.214,E2 -7428.214} C_VEL
LIN {X 0,Y 474.614,Z 229.367,A -85,B 0,C 180,E1 -7431.542,E2 -7431.542} C_VEL
LIN {X 0,Y 474.532,Z 229.376,A -85,B 0,C 180,E1 -7434.717,E2 -7434.717} C_VEL
LIN {X 0,Y 474.212,Z 229.561,A -85,B 0,C 180,E1 -7437.647,E2 -7437.647} C_VEL
LIN {X 0,Y 474.15,Z 232.874,A -85,B 0,C 180,E1 -7440.988,E2 -7440.988} C_VEL
LIN {X 0,Y 474.063,Z 235.503,A -85,B 0,C 180,E1 -7443.592,E2 -7443.592} C_VEL
LIN {X 0,Y 474.017,Z 238.376,A -85,B 0,C 180,E1 -7446.402,E2 -7446.402} C_VEL
LIN {X 0,Y 473.972,Z 241.247,A -85,B 0,C 180,E1 -7449.153,E2 -7449.153} C_VEL
LIN {X 0,Y 473.956,Z 243.846,A -85,B 0,C 180,E1 -7451.506,E2 -7451.506} C_VEL
LIN {X 0,Y 473.289,Z 244.445,A -85,B 0,C 180,E1 -7451.973,E2 -7451.973} C_VEL
LIN {X 0,Y 470.424,Z 245.572,A -85,B 0,C 180,E1 -7452.7,E2 -7452.7} C_VEL
LIN {X 0,Y 467.542,Z 246.723,A -85,B 0,C 180,E1 -7453.434,E2 -7453.434} C_VEL
LIN {X 0,Y 466.87,Z 247.359,A -85,B 0,C 180,E1 -7453.911,E2 -7453.911} C_VEL
LIN {X 0,Y 466.947,Z 248.289,A -85,B 0,C 180,E1 -7454.682,E2 -7454.682} C_VEL
LIN {X 0,Y 470.357,Z 263.267,A -85,B 0,C 180,E1 -7455.27,E2 -7455.27} C_VEL
LIN {X 0,Y 470.125,Z 275.534,A -85,B 0,C 180,E1 -7455.83,E2 -7455.83} C_VEL
LIN {X 0,Y 469.698,Z 287.418,A -85,B 0,C 180,E1 -7456.553,E2 -7456.553} C_VEL
LIN {X 0,Y 469.193,Z 298.974,A -85,B 0,C 180,E1 -7457.455,E2 -7457.455} C_VEL
LIN {X 0,Y 468.773,Z 307.9,A -85,B 0,C 180,E1 -7458.323,E2 -7458.323} C_VEL
LIN {X 0,Y 468.317,Z 317.052,A -85,B 0,C 180,E1 -7459.407,E2 -7459.407} C_VEL
LIN {X 0,Y 467.853,Z 325.93,A -85,B 0,C 180,E1 -7460.707,E2 -7460.707} C_VEL
LIN {X 0,Y 467.466,Z 333.074,A -85,B 0,C 180,E1 -7462.006,E2 -7462.006} C_VEL
LIN {X 0,Y 467.222,Z 339.164,A -85,B 0,C 180,E1 -7463.41,E2 -7463.41} C_VEL
LIN {X 0,Y 466.915,Z 343.879,A -85,B 0,C 180,E1 -7464.818,E2 -7464.818} C_VEL
LIN {X 0,Y 466.969,Z 346.143,A -85,B 0,C 180,E1 -7465.684,E2 -7465.684} C_VEL
LIN {X 0,Y 466.891,Z 347.994,A -85,B 0,C 180,E1 -7466.548,E2 -7466.548} C_VEL
LIN {X 0,Y 466.835,Z 349.389,A -85,B 0,C 180,E1 -7467.411,E2 -7467.411} C_VEL
LIN {X 0,Y 466.635,Z 351,A -85,B 0,C 180,E1 -7469.137,E2 -7469.137} C_VEL
LIN {X 0,Y 466.62,Z 351.234,A -85,B 0,C 180,E1 -7470,E2 -7470} C_VEL
LIN {X 0,Y 466.702,Z 350.467,A -85,B 0,C 180,E1 -7471.726,E2 -7471.726} C_VEL
LIN {X 0,Y 466.835,Z 349.503,A -85,B 0,C 180,E1 -7472.588,E2 -7472.588} C_VEL
LIN {X 0,Y 466.891,Z 348.158,A -85,B 0,C 180,E1 -7473.452,E2 -7473.452} C_VEL
LIN {X 0,Y 466.962,Z 345.316,A -85,B 0,C 180,E1 -7474.748,E2 -7474.748} C_VEL
LIN {X 0,Y 467.083,Z 341.46,A -85,B 0,C 180,E1 -7476.046,E2 -7476.046} C_VEL
LIN {X 0,Y 467.277,Z 336.481,A -85,B 0,C 180,E1 -7477.345,E2 -7477.345} C_VEL
LIN {X 0,Y 467.597,Z 330.209,A -85,B 0,C 180,E1 -7478.644,E2 -7478.644} C_VEL
LIN {X 0,Y 467.974,Z 322.352,A -85,B 0,C 180,E1 -7479.945,E2 -7479.945} C_VEL
LIN {X 0,Y 468.536,Z 312.568,A -85,B 0,C 180,E1 -7481.245,E2 -7481.245} C_VEL
LIN {X 0,Y 469.031,Z 302.3,A -85,B 0,C 180,E1 -7482.329,E2 -7482.329} C_VEL
LIN {X 0,Y 469.555,Z 290.632,A -85,B 0,C 180,E1 -7483.31,E2 -7483.31} C_VEL
LIN {X 0,Y 469.971,Z 279.164,A -85,B 0,C 180,E1 -7484.064,E2 -7484.064} C_VEL
LIN {X 0,Y 470.32,Z 267.151,A -85,B 0,C 180,E1 -7484.661,E2 -7484.661} C_VEL
LIN {X 0,Y 470.241,Z 262.692,A -85,B 0,C 180,E1 -7484.847,E2 -7484.847} C_VEL
LIN {X 0,Y 467.289,Z 249.977,A -85,B 0,C 180,E1 -7485.344,E2 -7485.344} C_VEL
LIN {X 0,Y 466.911,Z 248.227,A -85,B 0,C 180,E1 -7485.414,E2 -7485.414} C_VEL
LIN {X 0,Y 466.891,Z 244.646,A -85,B 0,C 180,E1 -7488.499,E2 -7488.499} C_VEL
LIN {X 0,Y 466.894,Z 241.697,A -85,B 0,C 180,E1 -7491.178,E2 -7491.178} C_VEL
LIN {X 0,Y 466.948,Z 238.768,A -85,B 0,C 180,E1 -7493.977,E2 -7493.977} C_VEL
LIN {X 0,Y 467.013,Z 235.842,A -85,B 0,C 180,E1 -7496.838,E2 -7496.838} C_VEL
LIN {X 0,Y 467.081,Z 232.95,A -85,B 0,C 180,E1 -7499.771,E2 -7499.771} C_VEL
LIN {X 0,Y 467.171,Z 230.295,A -85,B 0,C 180,E1 -7502.6,E2 -7502.6} C_VEL
LIN {X 0,Y 467.423,Z 230.262,A -85,B 0,C 180,E1 -7504.845,E2 -7504.845} C_VEL
LIN {X 0,Y 467.564,Z 230.243,A -85,B 0,C 180,E1 -7508.045,E2 -7508.045} C_VEL
LIN {X 0,Y 467.577,Z 230.241,A -85,B 0,C 180,E1 -7511.276,E2 -7511.276} C_VEL
LIN {X 0,Y 467.548,Z 230.246,A -85,B 0,C 180,E1 -7513.82,E2 -7513.82} C_VEL
LIN {X 0,Y 467.55,Z 230.245,A -85,B 0,C 180,E1 -7516.255,E2 -7516.255} C_VEL
LIN {X 0,Y 467.572,Z 230.243,A -85,B 0,C 180,E1 -7519.735,E2 -7519.735} C_VEL
LIN {X 0,Y 467.55,Z 230.245,A -85,B 0,C 180,E1 -7522.814,E2 -7522.814} C_VEL
LIN {X 0,Y 467.58,Z 230.244,A -85,B 0,C 180,E1 -7525.76,E2 -7525.76} C_VEL
LIN {X 0,Y 467.568,Z 230.241,A -85,B 0,C 180,E1 -7528.956,E2 -7528.956} C_VEL
LIN {X 0,Y 467.564,Z 230.243,A -85,B 0,C 180,E1 -7532.227,E2 -7532.227} C_VEL
LIN {X 0,Y 467.586,Z 230.242,A -85,B 0,C 180,E1 -7535.112,E2 -7535.112} C_VEL
LIN {X 0,Y 467.538,Z 230.247,A -85,B 0,C 180,E1 -7537.926,E2 -7537.926} C_VEL
LIN {X 0,Y 467.623,Z 230.235,A -85,B 0,C 180,E1 -7540.692,E2 -7540.692} C_VEL
LIN {X 0,Y 467.64,Z 230.232,A -85,B 0,C 180,E1 -7544.305,E2 -7544.305} C_VEL
LIN {X 0,Y 467.66,Z 230.231,A -85,B 0,C 180,E1 -7547.855,E2 -7547.855} C_VEL
LIN {X 0,Y 467.684,Z 230.23,A -85,B 0,C 180,E1 -7551.357,E2 -7551.357} C_VEL
LIN {X 0,Y 467.736,Z 230.221,A -85,B 0,C 180,E1 -7553.962,E2 -7553.962} C_VEL
LIN {X 0,Y 467.825,Z 230.208,A -85,B 0,C 180,E1 -7557.417,E2 -7557.417} C_VEL
LIN {X 0,Y 467.852,Z 230.207,A -85,B 0,C 180,E1 -7560,E2 -7560} C_VEL
LIN {X 0,Y 467.862,Z 230.206,A -85,B 0,C 180,E1 -7562.583,E2 -7562.583} C_VEL
LIN {X 0,Y 467.738,Z 230.222,A -85,B 0,C 180,E1 -7566.037,E2 -7566.037} C_VEL
LIN {X 0,Y 467.669,Z 230.232,A -85,B 0,C 180,E1 -7568.643,E2 -7568.643} C_VEL
LIN {X 0,Y 467.65,Z 230.234,A -85,B 0,C 180,E1 -7572.354,E2 -7572.354} C_VEL
LIN {X 0,Y 467.653,Z 230.234,A -85,B 0,C 180,E1 -7575.885,E2 -7575.885} C_VEL
LIN {X 0,Y 467.626,Z 230.236,A -85,B 0,C 180,E1 -7579.308,E2 -7579.308} C_VEL
LIN {X 0,Y 467.537,Z 230.249,A -85,B 0,C 180,E1 -7582.074,E2 -7582.074} C_VEL
LIN {X 0,Y 467.561,Z 230.241,A -85,B 0,C 180,E1 -7584.89,E2 -7584.89} C_VEL
LIN {X 0,Y 467.547,Z 230.247,A -85,B 0,C 180,E1 -7587.774,E2 -7587.774} C_VEL
LIN {X 0,Y 467.568,Z 230.244,A -85,B 0,C 180,E1 -7591.044,E2 -7591.044} C_VEL
LIN {X 0,Y 467.59,Z 230.24,A -85,B 0,C 180,E1 -7594.242,E2 -7594.242} C_VEL
LIN {X 0,Y 467.544,Z 230.246,A -85,B 0,C 180,E1 -7597.185,E2 -7597.185} C_VEL
LIN {X 0,Y 467.56,Z 230.241,A -85,B 0,C 180,E1 -7600.267,E2 -7600.267} C_VEL
LIN {X 0,Y 467.548,Z 230.244,A -85,B 0,C 180,E1 -7603.745,E2 -7603.745} C_VEL
LIN {X 0,Y 467.556,Z 230.247,A -85,B 0,C 180,E1 -7606.255,E2 -7606.255} C_VEL
LIN {X 0,Y 467.59,Z 230.279,A -85,B 0,C 180,E1 -7609.454,E2 -7609.454} C_VEL
LIN {X 0,Y 468.857,Z 237.409,A -85,B 0,C 180,E1 -7612.604,E2 -7612.604} C_VEL
LIN {X 0,Y 469.316,Z 241.436,A -85,B 0,C 180,E1 -7614.266,E2 -7614.266} C_VEL
LIN {X 0,Y 469.006,Z 248.679,A -85,B 0,C 180,E1 -7617.051,E2 -7617.051} C_VEL
LIN {X 0,Y 468.624,Z 256.222,A -85,B 0,C 180,E1 -7619.841,E2 -7619.841} C_VEL
